KUKA KRL program: EPS_2_251729_MH3A_A_20251114081656.src

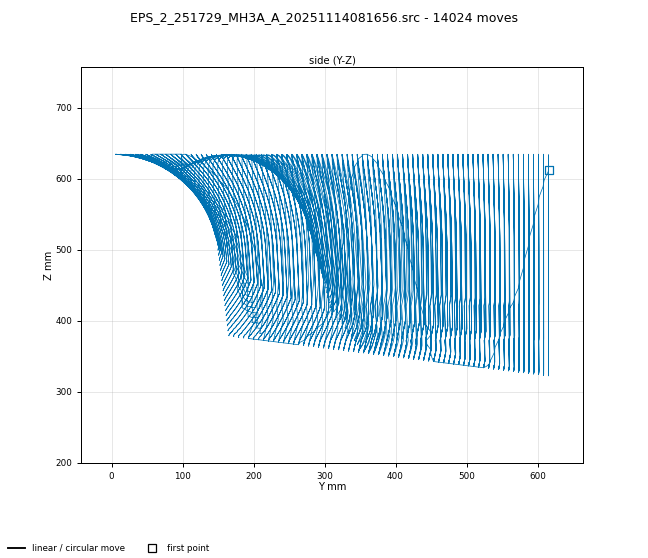
[picture p0: tool path of EPS_2_251729_MH3A_A_20251114081656.src, 14024 of 14026 moves have a stored position in this frame; points joined in program order, loops and branches not executed]
&ACCESS RVP
&REL 4
&COMMENT QRS 19112012
&PARAM EDITMASK = *
DEF PART()
EXT BAS (BAS_COMMAND :IN,REAL :IN )
INT I
BAS (#INITMOV,0 )

;KUKA QRS Post kuka4.cps  Date:22-06-2017 !

File_ID=2916

QRS_PRE_INIT()

;Init var - Until changes are made in qrs_pre_init
Outlet_Square_prg=0
Inlet_1_Square_prg=0
Inlet_2_Square_prg=0
Inlet_3_Square_prg=0
Inlet_4_Square_prg=0
Inlet_5_Square_prg=0

Outlet_1={X 0.000, Y 527.380, Z 509.000, B 0.000, E1 0.000 }
Inlet_1={X 0.000, Y 530.110, Z 534.000, B 0.000, E1 90.000 }
Inlet_2={X 0.000, Y 527.380, Z 509.000, B 0.000, E1 180.000 }
Outlet_1_type=251
Inlet_1_type=201
Inlet_2_type=251
;QRS#1=Sidecore dimensions
;QRS#2=250-10" PVC SDR 35
;QRS#3=200-8" PVC SDR 35
;QRS#4=250-10" PVC SDR 35
;QRS#5=
;QRS#6=
;QRS#7=
;QRS#8=
;QRS#9=14M PSX
;QRS#10=12-08 PSX
;QRS#11=14M PSX
;QRS#12=
;QRS#13=
;QRS#14=
;QRS#15=
;QRS#16=1220x127x914 3'
;QRS#17=EPS Height
;QRS#18=634,5
;QRS#19=*
;QRS#20= UPDATED VERSION 22-06-2017
;QRS#21=*
Outlet_Square=0100
Inlet_1_Square=0100
Inlet_2_Square=0100
Inlet_3_Square=0
Inlet_4_Square=0
Inlet_5_Square=0
Mill_Square=1
Outlet_Square_Prg=205
Inlet_1_Square_prg=204
Inlet_2_Square_prg=205

QRS_INIT()

$ADVANCE=5

; T1
PTP {E1 173.417,E2 173.417}
PTP {X 0,Y 615.497,A -85,B 0,C 180,E1 173.417,E2 173.417,E3 0,E4 0,E5 0,E6 0}
QRS_SPEED_INIT()
LIN {X 0,Y 615.497,Z 612.701,A -85,B 0,C 180,E1 173.417,E2 173.417,E3 0,E4 0,E5 0,E6 0} C_VEL
LIN {X 0,Y 615.497,Z 605.036,A -85,B 0,C 180,E1 172.455,E2 172.455} C_VEL
LIN {X 0,Y 615.498,Z 595.258,A -85,B 0,C 180,E1 171.463,E2 171.463} C_VEL
LIN {X 0,Y 615.497,Z 584.992,A -85,B 0,C 180,E1 170.636,E2 170.636} C_VEL
LIN {X 0,Y 615.479,Z 573.43,A -85,B 0,C 180,E1 169.888,E2 169.888} C_VEL
LIN {X 0,Y 615.499,Z 561.522,A -85,B 0,C 180,E1 169.291,E2 169.291} C_VEL
LIN {X 0,Y 615.498,Z 548.655,A -85,B 0,C 180,E1 168.807,E2 168.807} C_VEL
LIN {X 0,Y 615.493,Z 536.054,A -85,B 0,C 180,E1 168.473,E2 168.473} C_VEL
LIN {X 0,Y 615.488,Z 522.928,A -85,B 0,C 180,E1 168.264,E2 168.264} C_VEL
LIN {X 0,Y 615.497,Z 421.645,A -85,B 0,C 180,E1 167.072,E2 167.072} C_VEL
LIN {X 0,Y 615.491,Z 420.224,A -85,B 0,C 180,E1 166.967,E2 166.967} C_VEL
LIN {X 0,Y 615.492,Z 395.066,A -85,B 0,C 180,E1 164.095,E2 164.095} C_VEL
LIN {X 0,Y 615.492,Z 371.363,A -85,B 0,C 180,E1 161.354,E2 161.354} C_VEL
LIN {X 0,Y 615.498,Z 347.631,A -85,B 0,C 180,E1 158.568,E2 158.568} C_VEL
LIN {X 0,Y 615.497,Z 323.889,A -85,B 0,C 180,E1 155.728,E2 155.728} C_VEL
LIN {X 0,Y 615.495,Z 322.471,A -85,B 0,C 180,E1 155.504,E2 155.504} C_VEL
LIN {X 0,Y 615.484,Z 322.311,A -85,B 0,C 180,E1 152.823,E2 152.823} C_VEL
LIN {X 0,Y 615.477,Z 322.312,A -85,B 0,C 180,E1 150.208,E2 150.208} C_VEL
LIN {X 0,Y 615.495,Z 322.325,A -85,B 0,C 180,E1 147.543,E2 147.543} C_VEL
LIN {X 0,Y 615.481,Z 322.316,A -85,B 0,C 180,E1 145.184,E2 145.184} C_VEL
LIN {X 0,Y 615.489,Z 322.307,A -85,B 0,C 180,E1 142.758,E2 142.758} C_VEL
LIN {X 0,Y 615.485,Z 322.321,A -85,B 0,C 180,E1 139.912,E2 139.912} C_VEL
LIN {X 0,Y 615.491,Z 322.323,A -85,B 0,C 180,E1 137.647,E2 137.647} C_VEL
LIN {X 0,Y 615.48,Z 322.31,A -85,B 0,C 180,E1 134.931,E2 134.931} C_VEL
LIN {X 0,Y 615.485,Z 322.32,A -85,B 0,C 180,E1 132.08,E2 132.08} C_VEL
LIN {X 0,Y 615.494,Z 322.321,A -85,B 0,C 180,E1 129.75,E2 129.75} C_VEL
LIN {X 0,Y 615.483,Z 322.309,A -85,B 0,C 180,E1 126.936,E2 126.936} C_VEL
LIN {X 0,Y 615.494,Z 322.326,A -85,B 0,C 180,E1 124.022,E2 124.022} C_VEL
LIN {X 0,Y 615.488,Z 322.316,A -85,B 0,C 180,E1 121.686,E2 121.686} C_VEL
LIN {X 0,Y 615.477,Z 322.312,A -85,B 0,C 180,E1 119.407,E2 119.407} C_VEL
LIN {X 0,Y 615.486,Z 322.308,A -85,B 0,C 180,E1 117.044,E2 117.044} C_VEL
LIN {X 0,Y 615.491,Z 322.324,A -85,B 0,C 180,E1 114.273,E2 114.273} C_VEL
LIN {X 0,Y 615.495,Z 322.53,A -85,B 0,C 180,E1 112.137,E2 112.137} C_VEL
LIN {X 0,Y 615.495,Z 339.273,A -85,B 0,C 180,E1 109.859,E2 109.859} C_VEL
LIN {X 0,Y 615.493,Z 361.461,A -85,B 0,C 180,E1 106.929,E2 106.929} C_VEL
LIN {X 0,Y 615.479,Z 372.134,A -85,B 0,C 180,E1 105.566,E2 105.566} C_VEL
LIN {X 0,Y 615.477,Z 377.127,A -85,B 0,C 180,E1 105.481,E2 105.481} C_VEL
LIN {X 0,Y 615.498,Z 509.136,A -85,B 0,C 180,E1 103.905,E2 103.905} C_VEL
LIN {X 0,Y 615.497,Z 522.72,A -85,B 0,C 180,E1 103.622,E2 103.622} C_VEL
LIN {X 0,Y 615.497,Z 536.468,A -85,B 0,C 180,E1 103.202,E2 103.202} C_VEL
LIN {X 0,Y 615.493,Z 548.884,A -85,B 0,C 180,E1 102.698,E2 102.698} C_VEL
LIN {X 0,Y 615.496,Z 561.829,A -85,B 0,C 180,E1 102.029,E2 102.029} C_VEL
LIN {X 0,Y 615.499,Z 573.548,A -85,B 0,C 180,E1 101.277,E2 101.277} C_VEL
LIN {X 0,Y 615.498,Z 585.217,A -85,B 0,C 180,E1 100.361,E2 100.361} C_VEL
LIN {X 0,Y 615.497,Z 595.643,A -85,B 0,C 180,E1 99.365,E2 99.365} C_VEL
LIN {X 0,Y 615.496,Z 604.233,A -85,B 0,C 180,E1 98.372,E2 98.372} C_VEL
LIN {X 0,Y 615.495,Z 612.448,A -85,B 0,C 180,E1 97.216,E2 97.216} C_VEL
LIN {X 0,Y 615.496,Z 618.179,A -85,B 0,C 180,E1 96.228,E2 96.228} C_VEL
LIN {X 0,Y 615.491,Z 622.885,A -85,B 0,C 180,E1 95.242,E2 95.242} C_VEL
LIN {X 0,Y 615.496,Z 627.754,A -85,B 0,C 180,E1 93.929,E2 93.929} C_VEL
LIN {X 0,Y 615.496,Z 631.152,A -85,B 0,C 180,E1 92.619,E2 92.619} C_VEL
LIN {X 0,Y 615.493,Z 633.173,A -85,B 0,C 180,E1 91.309,E2 91.309} C_VEL
LIN {X 0,Y 615.494,Z 633.884,A -85,B 0,C 180,E1 90.001,E2 90.001} C_VEL
LIN {X 0,Y 615.49,Z 633.281,A -85,B 0,C 180,E1 88.692,E2 88.692} C_VEL
LIN {X 0,Y 615.493,Z 631.352,A -85,B 0,C 180,E1 87.383,E2 87.383} C_VEL
LIN {X 0,Y 615.496,Z 628.048,A -85,B 0,C 180,E1 86.072,E2 86.072} C_VEL
LIN {X 0,Y 615.496,Z 623.277,A -85,B 0,C 180,E1 84.76,E2 84.76} C_VEL
LIN {X 0,Y 615.494,Z 616.879,A -85,B 0,C 180,E1 83.444,E2 83.444} C_VEL
LIN {X 0,Y 615.496,Z 609.75,A -85,B 0,C 180,E1 82.29,E2 82.29} C_VEL
LIN {X 0,Y 615.497,Z 602.278,A -85,B 0,C 180,E1 81.299,E2 81.299} C_VEL
LIN {X 0,Y 615.495,Z 593.3,A -85,B 0,C 180,E1 80.305,E2 80.305} C_VEL
LIN {X 0,Y 615.499,Z 582.211,A -85,B 0,C 180,E1 79.291,E2 79.291} C_VEL
LIN {X 0,Y 615.498,Z 571.294,A -85,B 0,C 180,E1 78.474,E2 78.474} C_VEL
LIN {X 0,Y 615.489,Z 559,A -85,B 0,C 180,E1 77.722,E2 77.722} C_VEL
LIN {X 0,Y 615.498,Z 547.167,A -85,B 0,C 180,E1 77.136,E2 77.136} C_VEL
LIN {X 0,Y 615.493,Z 534.248,A -85,B 0,C 180,E1 76.632,E2 76.632} C_VEL
LIN {X 0,Y 615.498,Z 521.28,A -85,B 0,C 180,E1 76.253,E2 76.253} C_VEL
LIN {X 0,Y 615.497,Z 507.999,A -85,B 0,C 180,E1 75.988,E2 75.988} C_VEL
LIN {X 0,Y 615.481,Z 372.767,A -85,B 0,C 180,E1 74.372,E2 74.372} C_VEL
LIN {X 0,Y 615.486,Z 371.322,A -85,B 0,C 180,E1 74.266,E2 74.266} C_VEL
LIN {X 0,Y 615.477,Z 350.657,A -85,B 0,C 180,E1 71.559,E2 71.559} C_VEL
LIN {X 0,Y 615.493,Z 329.507,A -85,B 0,C 180,E1 68.745,E2 68.745} C_VEL
LIN {X 0,Y 615.494,Z 322.495,A -85,B 0,C 180,E1 67.759,E2 67.759} C_VEL
LIN {X 0,Y 615.488,Z 322.309,A -85,B 0,C 180,E1 65.009,E2 65.009} C_VEL
LIN {X 0,Y 615.48,Z 322.309,A -85,B 0,C 180,E1 62.824,E2 62.824} C_VEL
LIN {X 0,Y 615.497,Z 322.313,A -85,B 0,C 180,E1 60.204,E2 60.204} C_VEL
LIN {X 0,Y 615.489,Z 322.316,A -85,B 0,C 180,E1 57.544,E2 57.544} C_VEL
LIN {X 0,Y 615.499,Z 322.306,A -85,B 0,C 180,E1 55.187,E2 55.187} C_VEL
LIN {X 0,Y 615.477,Z 322.311,A -85,B 0,C 180,E1 52.759,E2 52.759} C_VEL
LIN {X 0,Y 615.493,Z 322.322,A -85,B 0,C 180,E1 49.911,E2 49.911} C_VEL
LIN {X 0,Y 615.481,Z 322.309,A -85,B 0,C 180,E1 46.953,E2 46.953} C_VEL
LIN {X 0,Y 615.486,Z 322.323,A -85,B 0,C 180,E1 43.999,E2 43.999} C_VEL
LIN {X 0,Y 615.487,Z 322.309,A -85,B 0,C 180,E1 41.474,E2 41.474} C_VEL
LIN {X 0,Y 615.478,Z 322.312,A -85,B 0,C 180,E1 38.905,E2 38.905} C_VEL
LIN {X 0,Y 615.489,Z 322.322,A -85,B 0,C 180,E1 36.425,E2 36.425} C_VEL
LIN {X 0,Y 615.484,Z 322.309,A -85,B 0,C 180,E1 33.536,E2 33.536} C_VEL
LIN {X 0,Y 615.48,Z 322.314,A -85,B 0,C 180,E1 30.92,E2 30.92} C_VEL
LIN {X 0,Y 615.498,Z 322.325,A -85,B 0,C 180,E1 28.455,E2 28.455} C_VEL
LIN {X 0,Y 615.484,Z 322.308,A -85,B 0,C 180,E1 25.571,E2 25.571} C_VEL
LIN {X 0,Y 615.484,Z 322.318,A -85,B 0,C 180,E1 22.845,E2 22.845} C_VEL
LIN {X 0,Y 615.479,Z 322.313,A -85,B 0,C 180,E1 20.033,E2 20.033} C_VEL
LIN {X 0,Y 615.493,Z 322.309,A -85,B 0,C 180,E1 17.27,E2 17.27} C_VEL
LIN {X 0,Y 615.496,Z 322.32,A -85,B 0,C 180,E1 14.549,E2 14.549} C_VEL
LIN {X 0,Y 615.476,Z 322.311,A -85,B 0,C 180,E1 11.861,E2 11.861} C_VEL
LIN {X 0,Y 615.487,Z 322.315,A -85,B 0,C 180,E1 9.199,E2 9.199} C_VEL
LIN {X 0,Y 615.498,Z 322.315,A -85,B 0,C 180,E1 6.557,E2 6.557} C_VEL
LIN {X 0,Y 615.476,Z 322.31,A -85,B 0,C 180,E1 3.929,E2 3.929} C_VEL
LIN {X 0,Y 615.494,Z 322.315,A -85,B 0,C 180,E1 1.309,E2 1.309} C_VEL
LIN {X 0,Y 615.495,Z 322.316,A -85,B 0,C 180,E1 -1.309,E2 -1.309} C_VEL
LIN {X 0,Y 615.476,Z 322.31,A -85,B 0,C 180,E1 -3.929,E2 -3.929} C_VEL
LIN {X 0,Y 615.496,Z 322.316,A -85,B 0,C 180,E1 -6.597,E2 -6.597} C_VEL
LIN {X 0,Y 615.488,Z 322.316,A -85,B 0,C 180,E1 -9.199,E2 -9.199} C_VEL
LIN {X 0,Y 615.478,Z 322.31,A -85,B 0,C 180,E1 -11.861,E2 -11.861} C_VEL
LIN {X 0,Y 615.497,Z 322.319,A -85,B 0,C 180,E1 -14.549,E2 -14.549} C_VEL
LIN {X 0,Y 615.493,Z 322.31,A -85,B 0,C 180,E1 -17.27,E2 -17.27} C_VEL
LIN {X 0,Y 615.479,Z 322.313,A -85,B 0,C 180,E1 -20.033,E2 -20.033} C_VEL
LIN {X 0,Y 615.487,Z 322.319,A -85,B 0,C 180,E1 -22.845,E2 -22.845} C_VEL
LIN {X 0,Y 615.484,Z 322.308,A -85,B 0,C 180,E1 -25.571,E2 -25.571} C_VEL
LIN {X 0,Y 615.497,Z 322.325,A -85,B 0,C 180,E1 -28.455,E2 -28.455} C_VEL
LIN {X 0,Y 615.486,Z 322.31,A -85,B 0,C 180,E1 -31.088,E2 -31.088} C_VEL
LIN {X 0,Y 615.484,Z 322.309,A -85,B 0,C 180,E1 -33.536,E2 -33.536} C_VEL
LIN {X 0,Y 615.488,Z 322.324,A -85,B 0,C 180,E1 -36.425,E2 -36.425} C_VEL
LIN {X 0,Y 615.481,Z 322.31,A -85,B 0,C 180,E1 -39.063,E2 -39.063} C_VEL
LIN {X 0,Y 615.486,Z 322.309,A -85,B 0,C 180,E1 -41.474,E2 -41.474} C_VEL
LIN {X 0,Y 615.497,Z 322.325,A -85,B 0,C 180,E1 -44.149,E2 -44.149} C_VEL
LIN {X 0,Y 615.481,Z 322.31,A -85,B 0,C 180,E1 -46.953,E2 -46.953} C_VEL
LIN {X 0,Y 615.485,Z 322.31,A -85,B 0,C 180,E1 -49.395,E2 -49.395} C_VEL
LIN {X 0,Y 615.49,Z 322.326,A -85,B 0,C 180,E1 -51.988,E2 -51.988} C_VEL
LIN {X 0,Y 615.486,Z 322.315,A -85,B 0,C 180,E1 -54.385,E2 -54.385} C_VEL
LIN {X 0,Y 615.478,Z 322.31,A -85,B 0,C 180,E1 -56.765,E2 -56.765} C_VEL
LIN {X 0,Y 615.492,Z 322.307,A -85,B 0,C 180,E1 -59.082,E2 -59.082} C_VEL
LIN {X 0,Y 615.489,Z 322.317,A -85,B 0,C 180,E1 -61.55,E2 -61.55} C_VEL
LIN {X 0,Y 615.481,Z 322.312,A -85,B 0,C 180,E1 -64.433,E2 -64.433} C_VEL
LIN {X 0,Y 615.49,Z 322.311,A -85,B 0,C 180,E1 -67.157,E2 -67.157} C_VEL
LIN {X 0,Y 615.494,Z 322.613,A -85,B 0,C 180,E1 -67.838,E2 -67.838} C_VEL
LIN {X 0,Y 615.491,Z 340.931,A -85,B 0,C 180,E1 -70.316,E2 -70.316} C_VEL
LIN {X 0,Y 615.493,Z 361.818,A -85,B 0,C 180,E1 -73.073,E2 -73.073} C_VEL
LIN {X 0,Y 615.481,Z 371.9,A -85,B 0,C 180,E1 -74.372,E2 -74.372} C_VEL
LIN {X 0,Y 615.479,Z 373.911,A -85,B 0,C 180,E1 -74.435,E2 -74.435} C_VEL
LIN {X 0,Y 615.5,Z 509.9,A -85,B 0,C 180,E1 -76.063,E2 -76.063} C_VEL
LIN {X 0,Y 615.497,Z 524.411,A -85,B 0,C 180,E1 -76.38,E2 -76.38} C_VEL
LIN {X 0,Y 615.497,Z 537.713,A -85,B 0,C 180,E1 -76.8,E2 -76.8} C_VEL
LIN {X 0,Y 615.497,Z 549.856,A -85,B 0,C 180,E1 -77.303,E2 -77.303} C_VEL
LIN {X 0,Y 615.493,Z 562.615,A -85,B 0,C 180,E1 -77.973,E2 -77.973} C_VEL
LIN {X 0,Y 615.499,Z 575.353,A -85,B 0,C 180,E1 -78.808,E2 -78.808} C_VEL
LIN {X 0,Y 615.498,Z 585.759,A -85,B 0,C 180,E1 -79.641,E2 -79.641} C_VEL
LIN {X 0,Y 615.496,Z 596.097,A -85,B 0,C 180,E1 -80.637,E2 -80.637} C_VEL
LIN {X 0,Y 615.497,Z 604.61,A -85,B 0,C 180,E1 -81.63,E2 -81.63} C_VEL
LIN {X 0,Y 615.496,Z 612.732,A -85,B 0,C 180,E1 -82.785,E2 -82.785} C_VEL
LIN {X 0,Y 615.496,Z 618.435,A -85,B 0,C 180,E1 -83.773,E2 -83.773} C_VEL
LIN {X 0,Y 615.495,Z 623.084,A -85,B 0,C 180,E1 -84.76,E2 -84.76} C_VEL
LIN {X 0,Y 615.494,Z 627.904,A -85,B 0,C 180,E1 -86.072,E2 -86.072} C_VEL
LIN {X 0,Y 615.496,Z 631.254,A -85,B 0,C 180,E1 -87.383,E2 -87.383} C_VEL
LIN {X 0,Y 615.489,Z 633.23,A -85,B 0,C 180,E1 -88.692,E2 -88.692} C_VEL
LIN {X 0,Y 615.493,Z 633.889,A -85,B 0,C 180,E1 -90.001,E2 -90.001} C_VEL
LIN {X 0,Y 615.489,Z 633.228,A -85,B 0,C 180,E1 -91.309,E2 -91.309} C_VEL
LIN {X 0,Y 615.496,Z 631.25,A -85,B 0,C 180,E1 -92.619,E2 -92.619} C_VEL
LIN {X 0,Y 615.494,Z 627.899,A -85,B 0,C 180,E1 -93.929,E2 -93.929} C_VEL
LIN {X 0,Y 615.495,Z 623.077,A -85,B 0,C 180,E1 -95.242,E2 -95.242} C_VEL
LIN {X 0,Y 615.496,Z 616.624,A -85,B 0,C 180,E1 -96.557,E2 -96.557} C_VEL
LIN {X 0,Y 615.497,Z 609.435,A -85,B 0,C 180,E1 -97.711,E2 -97.711} C_VEL
LIN {X 0,Y 615.497,Z 601.897,A -85,B 0,C 180,E1 -98.703,E2 -98.703} C_VEL
LIN {X 0,Y 615.495,Z 592.845,A -85,B 0,C 180,E1 -99.697,E2 -99.697} C_VEL
LIN {X 0,Y 615.497,Z 582.751,A -85,B 0,C 180,E1 -100.619,E2 -100.619} C_VEL
LIN {X 0,Y 615.498,Z 571.846,A -85,B 0,C 180,E1 -101.444,E2 -101.444} C_VEL
LIN {X 0,Y 615.488,Z 559.691,A -85,B 0,C 180,E1 -102.196,E2 -102.196} C_VEL
LIN {X 0,Y 615.498,Z 546.072,A -85,B 0,C 180,E1 -102.866,E2 -102.866} C_VEL
LIN {X 0,Y 615.497,Z 532.811,A -85,B 0,C 180,E1 -103.37,E2 -103.37} C_VEL
LIN {X 0,Y 615.498,Z 519.253,A -85,B 0,C 180,E1 -103.748,E2 -103.748} C_VEL
LIN {X 0,Y 615.497,Z 504.746,A -85,B 0,C 180,E1 -104.013,E2 -104.013} C_VEL
LIN {X 0,Y 615.48,Z 372.617,A -85,B 0,C 180,E1 -105.587,E2 -105.587} C_VEL
LIN {X 0,Y 615.486,Z 370.938,A -85,B 0,C 180,E1 -105.736,E2 -105.736} C_VEL
LIN {X 0,Y 615.477,Z 350.311,A -85,B 0,C 180,E1 -108.441,E2 -108.441} C_VEL
LIN {X 0,Y 615.496,Z 329.159,A -85,B 0,C 180,E1 -111.257,E2 -111.257} C_VEL
LIN {X 0,Y 615.494,Z 322.512,A -85,B 0,C 180,E1 -112.189,E2 -112.189} C_VEL
LIN {X 0,Y 615.492,Z 322.325,A -85,B 0,C 180,E1 -114.272,E2 -114.272} C_VEL
LIN {X 0,Y 615.486,Z 322.308,A -85,B 0,C 180,E1 -117.045,E2 -117.045} C_VEL
LIN {X 0,Y 615.497,Z 322.314,A -85,B 0,C 180,E1 -119.796,E2 -119.796} C_VEL
LIN {X 0,Y 615.488,Z 322.316,A -85,B 0,C 180,E1 -122.458,E2 -122.458} C_VEL
LIN {X 0,Y 615.499,Z 322.306,A -85,B 0,C 180,E1 -124.815,E2 -124.815} C_VEL
LIN {X 0,Y 615.477,Z 322.311,A -85,B 0,C 180,E1 -127.244,E2 -127.244} C_VEL
LIN {X 0,Y 615.492,Z 322.322,A -85,B 0,C 180,E1 -130.089,E2 -130.089} C_VEL
LIN {X 0,Y 615.481,Z 322.309,A -85,B 0,C 180,E1 -133.047,E2 -133.047} C_VEL
LIN {X 0,Y 615.486,Z 322.323,A -85,B 0,C 180,E1 -136.003,E2 -136.003} C_VEL
LIN {X 0,Y 615.487,Z 322.309,A -85,B 0,C 180,E1 -138.526,E2 -138.526} C_VEL
LIN {X 0,Y 615.478,Z 322.312,A -85,B 0,C 180,E1 -141.095,E2 -141.095} C_VEL
LIN {X 0,Y 615.489,Z 322.322,A -85,B 0,C 180,E1 -143.575,E2 -143.575} C_VEL
LIN {X 0,Y 615.484,Z 322.309,A -85,B 0,C 180,E1 -146.467,E2 -146.467} C_VEL
LIN {X 0,Y 615.48,Z 322.313,A -85,B 0,C 180,E1 -149.08,E2 -149.08} C_VEL
LIN {X 0,Y 615.497,Z 322.324,A -85,B 0,C 180,E1 -151.549,E2 -151.549} C_VEL
LIN {X 0,Y 615.484,Z 322.308,A -85,B 0,C 180,E1 -154.433,E2 -154.433} C_VEL
LIN {X 0,Y 615.499,Z 322.572,A -85,B 0,C 180,E1 -155.639,E2 -155.639} C_VEL
LIN {X 0,Y 615.479,Z 343.906,A -85,B 0,C 180,E1 -158.216,E2 -158.216} C_VEL
LIN {X 0,Y 615.484,Z 367.627,A -85,B 0,C 180,E1 -161.008,E2 -161.008} C_VEL
LIN {X 0,Y 615.483,Z 391.999,A -85,B 0,C 180,E1 -163.832,E2 -163.832} C_VEL
LIN {X 0,Y 615.491,Z 416.465,A -85,B 0,C 180,E1 -166.631,E2 -166.631} C_VEL
LIN {X 0,Y 615.495,Z 421.071,A -85,B 0,C 180,E1 -167.135,E2 -167.135} C_VEL
LIN {X 0,Y 615.491,Z 425.922,A -85,B 0,C 180,E1 -167.219,E2 -167.219} C_VEL
LIN {X 0,Y 615.486,Z 530.146,A -85,B 0,C 180,E1 -168.452,E2 -168.452} C_VEL
LIN {X 0,Y 615.499,Z 542.722,A -85,B 0,C 180,E1 -168.724,E2 -168.724} C_VEL
LIN {X 0,Y 615.497,Z 556.026,A -85,B 0,C 180,E1 -169.155,E2 -169.155} C_VEL
LIN {X 0,Y 615.491,Z 567.066,A -85,B 0,C 180,E1 -169.639,E2 -169.639} C_VEL
LIN {X 0,Y 615.482,Z 578.806,A -85,B 0,C 180,E1 -170.304,E2 -170.304} C_VEL
LIN {X 0,Y 615.499,Z 589.268,A -85,B 0,C 180,E1 -171.05,E2 -171.05} C_VEL
LIN {X 0,Y 615.498,Z 597.831,A -85,B 0,C 180,E1 -171.794,E2 -171.794} C_VEL
LIN {X 0,Y 615.498,Z 605.709,A -85,B 0,C 180,E1 -172.62,E2 -172.62} C_VEL
LIN {X 0,Y 615.497,Z 613.399,A -85,B 0,C 180,E1 -173.608,E2 -173.608} C_VEL
LIN {X 0,Y 615.498,Z 620.458,A -85,B 0,C 180,E1 -174.759,E2 -174.759} C_VEL
LIN {X 0,Y 615.493,Z 625.158,A -85,B 0,C 180,E1 -175.744,E2 -175.744} C_VEL
LIN {X 0,Y 615.496,Z 628.754,A -85,B 0,C 180,E1 -176.727,E2 -176.727} C_VEL
LIN {X 0,Y 615.496,Z 630.615,A -85,B 0,C 180,E1 -177.382,E2 -177.382} C_VEL
LIN {X 0,Y 615.497,Z 632.034,A -85,B 0,C 180,E1 -178.037,E2 -178.037} C_VEL
LIN {X 0,Y 615.496,Z 633.642,A -85,B 0,C 180,E1 -179.346,E2 -179.346} C_VEL
LIN {X 0,Y 615.494,Z 633.884,A -85,B 0,C 180,E1 -180,E2 -180} C_VEL
LIN {X 0,Y 615.496,Z 633.705,A -85,B 0,C 180,E1 -180.654,E2 -180.654} C_VEL
LIN {X 0,Y 615.496,Z 632.183,A -85,B 0,C 180,E1 -181.963,E2 -181.963} C_VEL
LIN {X 0,Y 615.498,Z 630.841,A -85,B 0,C 180,E1 -182.618,E2 -182.618} C_VEL
LIN {X 0,Y 615.497,Z 627.994,A -85,B 0,C 180,E1 -183.601,E2 -183.601} C_VEL
LIN {X 0,Y 615.499,Z 624.134,A -85,B 0,C 180,E1 -184.585,E2 -184.585} C_VEL
LIN {X 0,Y 615.498,Z 619.151,A -85,B 0,C 180,E1 -185.57,E2 -185.57} C_VEL
LIN {X 0,Y 615.497,Z 612.701,A -85,B 0,C 180,E1 -186.583,E2 -186.583} C_VEL
LIN {X 0,Y 614.829,Z 609.519,A -85,B 0,C 180,E1 -187.032,E2 -187.032} C_VEL
LIN {X 0,Y 611.988,Z 603.946,A -85,B 0,C 180,E1 -187.749,E2 -187.749} C_VEL
LIN {X 0,Y 609.138,Z 597.67,A -85,B 0,C 180,E1 -188.43,E2 -188.43} C_VEL
LIN {X 0,Y 608.477,Z 593.429,A -85,B 0,C 180,E1 -188.82,E2 -188.82} C_VEL
LIN {X 0,Y 608.489,Z 582.891,A -85,B 0,C 180,E1 -189.641,E2 -189.641} C_VEL
LIN {X 0,Y 608.49,Z 572.112,A -85,B 0,C 180,E1 -190.313,E2 -190.313} C_VEL
LIN {X 0,Y 608.515,Z 560.848,A -85,B 0,C 180,E1 -190.868,E2 -190.868} C_VEL
LIN {X 0,Y 608.534,Z 548.763,A -85,B 0,C 180,E1 -191.323,E2 -191.323} C_VEL
LIN {X 0,Y 608.542,Z 536.148,A -85,B 0,C 180,E1 -191.66,E2 -191.66} C_VEL
LIN {X 0,Y 608.539,Z 523.034,A -85,B 0,C 180,E1 -191.871,E2 -191.871} C_VEL
LIN {X 0,Y 608.556,Z 421.658,A -85,B 0,C 180,E1 -193.078,E2 -193.078} C_VEL
LIN {X 0,Y 608.48,Z 420.328,A -85,B 0,C 180,E1 -193.186,E2 -193.186} C_VEL
LIN {X 0,Y 608.533,Z 396.59,A -85,B 0,C 180,E1 -195.92,E2 -195.92} C_VEL
LIN {X 0,Y 608.546,Z 372.479,A -85,B 0,C 180,E1 -198.736,E2 -198.736} C_VEL
LIN {X 0,Y 608.623,Z 349.11,A -85,B 0,C 180,E1 -201.508,E2 -201.508} C_VEL
LIN {X 0,Y 608.674,Z 324.899,A -85,B 0,C 180,E1 -204.437,E2 -204.437} C_VEL
LIN {X 0,Y 608.49,Z 323.441,A -85,B 0,C 180,E1 -204.661,E2 -204.661} C_VEL
LIN {X 0,Y 608.447,Z 323.313,A -85,B 0,C 180,E1 -207.518,E2 -207.518} C_VEL
LIN {X 0,Y 608.462,Z 323.314,A -85,B 0,C 180,E1 -209.97,E2 -209.97} C_VEL
LIN {X 0,Y 608.463,Z 323.314,A -85,B 0,C 180,E1 -212.879,E2 -212.879} C_VEL
LIN {X 0,Y 608.439,Z 323.314,A -85,B 0,C 180,E1 -215.278,E2 -215.278} C_VEL
LIN {X 0,Y 608.468,Z 323.312,A -85,B 0,C 180,E1 -217.746,E2 -217.746} C_VEL
LIN {X 0,Y 608.448,Z 323.323,A -85,B 0,C 180,E1 -220.328,E2 -220.328} C_VEL
LIN {X 0,Y 608.484,Z 323.308,A -85,B 0,C 180,E1 -223.31,E2 -223.31} C_VEL
LIN {X 0,Y 608.469,Z 323.32,A -85,B 0,C 180,E1 -226.13,E2 -226.13} C_VEL
LIN {X 0,Y 608.45,Z 323.314,A -85,B 0,C 180,E1 -228.822,E2 -228.822} C_VEL
LIN {X 0,Y 608.469,Z 323.315,A -85,B 0,C 180,E1 -231.76,E2 -231.76} C_VEL
LIN {X 0,Y 608.449,Z 323.314,A -85,B 0,C 180,E1 -234.722,E2 -234.722} C_VEL
LIN {X 0,Y 608.462,Z 323.314,A -85,B 0,C 180,E1 -237.478,E2 -237.478} C_VEL
LIN {X 0,Y 608.481,Z 323.314,A -85,B 0,C 180,E1 -240.221,E2 -240.221} C_VEL
LIN {X 0,Y 608.477,Z 323.31,A -85,B 0,C 180,E1 -242.794,E2 -242.794} C_VEL
LIN {X 0,Y 608.457,Z 323.316,A -85,B 0,C 180,E1 -245.428,E2 -245.428} C_VEL
LIN {X 0,Y 608.493,Z 323.473,A -85,B 0,C 180,E1 -247.729,E2 -247.729} C_VEL
LIN {X 0,Y 608.574,Z 331.445,A -85,B 0,C 180,E1 -248.845,E2 -248.845} C_VEL
LIN {X 0,Y 608.511,Z 352.446,A -85,B 0,C 180,E1 -251.666,E2 -251.666} C_VEL
LIN {X 0,Y 608.531,Z 372.139,A -85,B 0,C 180,E1 -254.251,E2 -254.251} C_VEL
LIN {X 0,Y 608.647,Z 375.384,A -85,B 0,C 180,E1 -254.319,E2 -254.319} C_VEL
LIN {X 0,Y 608.61,Z 509.953,A -85,B 0,C 180,E1 -255.948,E2 -255.948} C_VEL
LIN {X 0,Y 608.613,Z 524.281,A -85,B 0,C 180,E1 -256.263,E2 -256.263} C_VEL
LIN {X 0,Y 608.586,Z 537.623,A -85,B 0,C 180,E1 -256.688,E2 -256.688} C_VEL
LIN {X 0,Y 608.544,Z 550.675,A -85,B 0,C 180,E1 -257.239,E2 -257.239} C_VEL
LIN {X 0,Y 608.536,Z 563.327,A -85,B 0,C 180,E1 -257.916,E2 -257.916} C_VEL
LIN {X 0,Y 608.5,Z 574.843,A -85,B 0,C 180,E1 -258.676,E2 -258.676} C_VEL
LIN {X 0,Y 608.495,Z 585.406,A -85,B 0,C 180,E1 -259.518,E2 -259.518} C_VEL
LIN {X 0,Y 608.48,Z 595.892,A -85,B 0,C 180,E1 -260.526,E2 -260.526} C_VEL
LIN {X 0,Y 608.463,Z 604.543,A -85,B 0,C 180,E1 -261.531,E2 -261.531} C_VEL
LIN {X 0,Y 608.461,Z 612.834,A -85,B 0,C 180,E1 -262.7,E2 -262.7} C_VEL
LIN {X 0,Y 608.443,Z 619.323,A -85,B 0,C 180,E1 -263.831,E2 -263.831} C_VEL
LIN {X 0,Y 608.437,Z 624.784,A -85,B 0,C 180,E1 -265.029,E2 -265.029} C_VEL
LIN {X 0,Y 608.434,Z 628.296,A -85,B 0,C 180,E1 -266.025,E2 -266.025} C_VEL
LIN {X 0,Y 608.424,Z 631.732,A -85,B 0,C 180,E1 -267.351,E2 -267.351} C_VEL
LIN {X 0,Y 608.446,Z 633.776,A -85,B 0,C 180,E1 -268.675,E2 -268.675} C_VEL
LIN {X 0,Y 608.434,Z 634.495,A -85,B 0,C 180,E1 -269.999,E2 -269.999} C_VEL
LIN {X 0,Y 608.443,Z 633.883,A -85,B 0,C 180,E1 -271.323,E2 -271.323} C_VEL
LIN {X 0,Y 608.421,Z 631.93,A -85,B 0,C 180,E1 -272.647,E2 -272.647} C_VEL
LIN {X 0,Y 608.434,Z 628.588,A -85,B 0,C 180,E1 -273.973,E2 -273.973} C_VEL
LIN {X 0,Y 608.44,Z 623.765,A -85,B 0,C 180,E1 -275.301,E2 -275.301} C_VEL
LIN {X 0,Y 608.438,Z 617.301,A -85,B 0,C 180,E1 -276.632,E2 -276.632} C_VEL
LIN {X 0,Y 608.453,Z 610.103,A -85,B 0,C 180,E1 -277.799,E2 -277.799} C_VEL
LIN {X 0,Y 608.476,Z 602.569,A -85,B 0,C 180,E1 -278.802,E2 -278.802} C_VEL
LIN {X 0,Y 608.486,Z 593.528,A -85,B 0,C 180,E1 -279.808,E2 -279.808} C_VEL
LIN {X 0,Y 608.507,Z 582.723,A -85,B 0,C 180,E1 -280.804,E2 -280.804} C_VEL
LIN {X 0,Y 608.523,Z 571.394,A -85,B 0,C 180,E1 -281.66,E2 -281.66} C_VEL
LIN {X 0,Y 608.54,Z 559.061,A -85,B 0,C 180,E1 -282.42,E2 -282.42} C_VEL
LIN {X 0,Y 608.56,Z 547.196,A -85,B 0,C 180,E1 -283.013,E2 -283.013} C_VEL
LIN {X 0,Y 608.581,Z 534.246,A -85,B 0,C 180,E1 -283.523,E2 -283.523} C_VEL
LIN {X 0,Y 608.593,Z 519.989,A -85,B 0,C 180,E1 -283.935,E2 -283.935} C_VEL
LIN {X 0,Y 608.614,Z 506.662,A -85,B 0,C 180,E1 -284.192,E2 -284.192} C_VEL
LIN {X 0,Y 608.587,Z 372.733,A -85,B 0,C 180,E1 -285.81,E2 -285.81} C_VEL
LIN {X 0,Y 608.498,Z 371.369,A -85,B 0,C 180,E1 -285.92,E2 -285.92} C_VEL
LIN {X 0,Y 608.524,Z 351.904,A -85,B 0,C 180,E1 -288.495,E2 -288.495} C_VEL
LIN {X 0,Y 608.571,Z 330.813,A -85,B 0,C 180,E1 -291.331,E2 -291.331} C_VEL
LIN {X 0,Y 608.495,Z 323.483,A -85,B 0,C 180,E1 -292.359,E2 -292.359} C_VEL
LIN {X 0,Y 608.457,Z 323.318,A -85,B 0,C 180,E1 -294.57,E2 -294.57} C_VEL
LIN {X 0,Y 608.475,Z 323.31,A -85,B 0,C 180,E1 -297.206,E2 -297.206} C_VEL
LIN {X 0,Y 608.477,Z 323.316,A -85,B 0,C 180,E1 -299.973,E2 -299.973} C_VEL
LIN {X 0,Y 608.463,Z 323.315,A -85,B 0,C 180,E1 -302.522,E2 -302.522} C_VEL
LIN {X 0,Y 608.447,Z 323.314,A -85,B 0,C 180,E1 -305.276,E2 -305.276} C_VEL
LIN {X 0,Y 608.471,Z 323.317,A -85,B 0,C 180,E1 -308.24,E2 -308.24} C_VEL
LIN {X 0,Y 608.477,Z 323.314,A -85,B 0,C 180,E1 -310.332,E2 -310.332} C_VEL
LIN {X 0,Y 608.465,Z 323.313,A -85,B 0,C 180,E1 -313.308,E2 -313.308} C_VEL
LIN {X 0,Y 608.471,Z 323.316,A -85,B 0,C 180,E1 -316.131,E2 -316.131} C_VEL
LIN {X 0,Y 608.452,Z 323.312,A -85,B 0,C 180,E1 -318.823,E2 -318.823} C_VEL
LIN {X 0,Y 608.464,Z 323.315,A -85,B 0,C 180,E1 -321.411,E2 -321.411} C_VEL
LIN {X 0,Y 608.47,Z 323.317,A -85,B 0,C 180,E1 -323.949,E2 -323.949} C_VEL
LIN {X 0,Y 608.46,Z 323.313,A -85,B 0,C 180,E1 -326.329,E2 -326.329} C_VEL
LIN {X 0,Y 608.471,Z 323.31,A -85,B 0,C 180,E1 -328.726,E2 -328.726} C_VEL
LIN {X 0,Y 608.476,Z 323.316,A -85,B 0,C 180,E1 -331.377,E2 -331.377} C_VEL
LIN {X 0,Y 608.445,Z 323.317,A -85,B 0,C 180,E1 -333.964,E2 -333.964} C_VEL
LIN {X 0,Y 608.461,Z 323.313,A -85,B 0,C 180,E1 -336.155,E2 -336.155} C_VEL
LIN {X 0,Y 608.47,Z 323.31,A -85,B 0,C 180,E1 -338.308,E2 -338.308} C_VEL
LIN {X 0,Y 608.471,Z 323.319,A -85,B 0,C 180,E1 -341.28,E2 -341.28} C_VEL
LIN {X 0,Y 608.457,Z 323.314,A -85,B 0,C 180,E1 -343.906,E2 -343.906} C_VEL
LIN {X 0,Y 608.463,Z 323.312,A -85,B 0,C 180,E1 -346.643,E2 -346.643} C_VEL
LIN {X 0,Y 608.474,Z 323.318,A -85,B 0,C 180,E1 -349.35,E2 -349.35} C_VEL
LIN {X 0,Y 608.471,Z 323.31,A -85,B 0,C 180,E1 -352.033,E2 -352.033} C_VEL
LIN {X 0,Y 608.469,Z 323.314,A -85,B 0,C 180,E1 -354.698,E2 -354.698} C_VEL
LIN {X 0,Y 608.485,Z 323.314,A -85,B 0,C 180,E1 -357.352,E2 -357.352} C_VEL
LIN {X 0,Y 608.468,Z 323.311,A -85,B 0,C 180,E1 -360,E2 -360} C_VEL
LIN {X 0,Y 608.485,Z 323.313,A -85,B 0,C 180,E1 -362.648,E2 -362.648} C_VEL
LIN {X 0,Y 608.47,Z 323.314,A -85,B 0,C 180,E1 -365.302,E2 -365.302} C_VEL
LIN {X 0,Y 608.471,Z 323.31,A -85,B 0,C 180,E1 -367.967,E2 -367.967} C_VEL
LIN {X 0,Y 608.473,Z 323.317,A -85,B 0,C 180,E1 -370.65,E2 -370.65} C_VEL
LIN {X 0,Y 608.464,Z 323.313,A -85,B 0,C 180,E1 -373.356,E2 -373.356} C_VEL
LIN {X 0,Y 608.457,Z 323.313,A -85,B 0,C 180,E1 -376.094,E2 -376.094} C_VEL
LIN {X 0,Y 608.455,Z 323.319,A -85,B 0,C 180,E1 -378.87,E2 -378.87} C_VEL
LIN {X 0,Y 608.47,Z 323.31,A -85,B 0,C 180,E1 -381.691,E2 -381.691} C_VEL
LIN {X 0,Y 608.452,Z 323.323,A -85,B 0,C 180,E1 -384.571,E2 -384.571} C_VEL
LIN {X 0,Y 608.475,Z 323.31,A -85,B 0,C 180,E1 -387.209,E2 -387.209} C_VEL
LIN {X 0,Y 608.46,Z 323.314,A -85,B 0,C 180,E1 -389.973,E2 -389.973} C_VEL
LIN {X 0,Y 608.467,Z 323.319,A -85,B 0,C 180,E1 -392.526,E2 -392.526} C_VEL
LIN {X 0,Y 608.437,Z 323.314,A -85,B 0,C 180,E1 -395.278,E2 -395.278} C_VEL
LIN {X 0,Y 608.467,Z 323.312,A -85,B 0,C 180,E1 -397.746,E2 -397.746} C_VEL
LIN {X 0,Y 608.474,Z 323.319,A -85,B 0,C 180,E1 -400.333,E2 -400.333} C_VEL
LIN {X 0,Y 608.483,Z 323.309,A -85,B 0,C 180,E1 -403.312,E2 -403.312} C_VEL
LIN {X 0,Y 608.467,Z 323.321,A -85,B 0,C 180,E1 -406.132,E2 -406.132} C_VEL
LIN {X 0,Y 608.45,Z 323.313,A -85,B 0,C 180,E1 -408.825,E2 -408.825} C_VEL
LIN {X 0,Y 608.47,Z 323.312,A -85,B 0,C 180,E1 -411.414,E2 -411.414} C_VEL
LIN {X 0,Y 608.476,Z 323.32,A -85,B 0,C 180,E1 -413.951,E2 -413.951} C_VEL
LIN {X 0,Y 608.464,Z 323.315,A -85,B 0,C 180,E1 -416.331,E2 -416.331} C_VEL
LIN {X 0,Y 608.474,Z 323.31,A -85,B 0,C 180,E1 -418.728,E2 -418.728} C_VEL
LIN {X 0,Y 608.476,Z 323.312,A -85,B 0,C 180,E1 -421.38,E2 -421.38} C_VEL
LIN {X 0,Y 608.471,Z 323.313,A -85,B 0,C 180,E1 -424.28,E2 -424.28} C_VEL
LIN {X 0,Y 608.45,Z 323.314,A -85,B 0,C 180,E1 -426.877,E2 -426.877} C_VEL
LIN {X 0,Y 608.505,Z 323.481,A -85,B 0,C 180,E1 -427.686,E2 -427.686} C_VEL
LIN {X 0,Y 608.57,Z 335.111,A -85,B 0,C 180,E1 -429.296,E2 -429.296} C_VEL
LIN {X 0,Y 608.546,Z 356.635,A -85,B 0,C 180,E1 -432.18,E2 -432.18} C_VEL
LIN {X 0,Y 608.541,Z 372.196,A -85,B 0,C 180,E1 -434.21,E2 -434.21} C_VEL
LIN {X 0,Y 608.66,Z 375.699,A -85,B 0,C 180,E1 -434.278,E2 -434.278} C_VEL
LIN {X 0,Y 608.62,Z 508.97,A -85,B 0,C 180,E1 -435.886,E2 -435.886} C_VEL
LIN {X 0,Y 608.595,Z 523.658,A -85,B 0,C 180,E1 -436.201,E2 -436.201} C_VEL
LIN {X 0,Y 608.584,Z 537.735,A -85,B 0,C 180,E1 -436.647,E2 -436.647} C_VEL
LIN {X 0,Y 608.564,Z 549.903,A -85,B 0,C 180,E1 -437.156,E2 -437.156} C_VEL
LIN {X 0,Y 608.516,Z 562.696,A -85,B 0,C 180,E1 -437.833,E2 -437.833} C_VEL
LIN {X 0,Y 608.499,Z 575.483,A -85,B 0,C 180,E1 -438.678,E2 -438.678} C_VEL
LIN {X 0,Y 608.495,Z 585.942,A -85,B 0,C 180,E1 -439.52,E2 -439.52} C_VEL
LIN {X 0,Y 608.479,Z 596.343,A -85,B 0,C 180,E1 -440.528,E2 -440.528} C_VEL
LIN {X 0,Y 608.464,Z 604.921,A -85,B 0,C 180,E1 -441.532,E2 -441.532} C_VEL
LIN {X 0,Y 608.461,Z 613.119,A -85,B 0,C 180,E1 -442.701,E2 -442.701} C_VEL
LIN {X 0,Y 608.443,Z 619.548,A -85,B 0,C 180,E1 -443.831,E2 -443.831} C_VEL
LIN {X 0,Y 608.438,Z 624.965,A -85,B 0,C 180,E1 -445.031,E2 -445.031} C_VEL
LIN {X 0,Y 608.431,Z 628.444,A -85,B 0,C 180,E1 -446.027,E2 -446.027} C_VEL
LIN {X 0,Y 608.424,Z 631.833,A -85,B 0,C 180,E1 -447.353,E2 -447.353} C_VEL
LIN {X 0,Y 608.442,Z 633.831,A -85,B 0,C 180,E1 -448.677,E2 -448.677} C_VEL
LIN {X 0,Y 608.433,Z 634.5,A -85,B 0,C 180,E1 -450.001,E2 -450.001} C_VEL
LIN {X 0,Y 608.442,Z 633.829,A -85,B 0,C 180,E1 -451.325,E2 -451.325} C_VEL
LIN {X 0,Y 608.424,Z 631.829,A -85,B 0,C 180,E1 -452.649,E2 -452.649} C_VEL
LIN {X 0,Y 608.431,Z 628.439,A -85,B 0,C 180,E1 -453.975,E2 -453.975} C_VEL
LIN {X 0,Y 608.44,Z 623.564,A -85,B 0,C 180,E1 -455.303,E2 -455.303} C_VEL
LIN {X 0,Y 608.446,Z 617.207,A -85,B 0,C 180,E1 -456.604,E2 -456.604} C_VEL
LIN {X 0,Y 608.453,Z 609.792,A -85,B 0,C 180,E1 -457.801,E2 -457.801} C_VEL
LIN {X 0,Y 608.473,Z 600.816,A -85,B 0,C 180,E1 -458.971,E2 -458.971} C_VEL
LIN {X 0,Y 608.472,Z 591.382,A -85,B 0,C 180,E1 -459.978,E2 -459.978} C_VEL
LIN {X 0,Y 608.506,Z 580.045,A -85,B 0,C 180,E1 -460.973,E2 -460.973} C_VEL
LIN {X 0,Y 608.533,Z 568.136,A -85,B 0,C 180,E1 -461.83,E2 -461.83} C_VEL
LIN {X 0,Y 608.53,Z 555.057,A -85,B 0,C 180,E1 -462.592,E2 -462.592} C_VEL
LIN {X 0,Y 608.563,Z 542.154,A -85,B 0,C 180,E1 -463.185,E2 -463.185} C_VEL
LIN {X 0,Y 608.597,Z 528.154,A -85,B 0,C 180,E1 -463.673,E2 -463.673} C_VEL
LIN {X 0,Y 608.624,Z 514.411,A -85,B 0,C 180,E1 -464.013,E2 -464.013} C_VEL
LIN {X 0,Y 608.624,Z 500.064,A -85,B 0,C 180,E1 -464.235,E2 -464.235} C_VEL
LIN {X 0,Y 608.558,Z 372.624,A -85,B 0,C 180,E1 -465.769,E2 -465.769} C_VEL
LIN {X 0,Y 608.496,Z 371.005,A -85,B 0,C 180,E1 -465.921,E2 -465.921} C_VEL
LIN {X 0,Y 608.524,Z 351.559,A -85,B 0,C 180,E1 -468.496,E2 -468.496} C_VEL
LIN {X 0,Y 608.574,Z 330.469,A -85,B 0,C 180,E1 -471.333,E2 -471.333} C_VEL
LIN {X 0,Y 608.506,Z 323.474,A -85,B 0,C 180,E1 -472.315,E2 -472.315} C_VEL
LIN {X 0,Y 608.458,Z 323.317,A -85,B 0,C 180,E1 -474.572,E2 -474.572} C_VEL
LIN {X 0,Y 608.476,Z 323.31,A -85,B 0,C 180,E1 -477.207,E2 -477.207} C_VEL
LIN {X 0,Y 608.476,Z 323.317,A -85,B 0,C 180,E1 -479.973,E2 -479.973} C_VEL
LIN {X 0,Y 608.455,Z 323.313,A -85,B 0,C 180,E1 -482.88,E2 -482.88} C_VEL
LIN {X 0,Y 608.447,Z 323.314,A -85,B 0,C 180,E1 -485.278,E2 -485.278} C_VEL
LIN {X 0,Y 608.472,Z 323.316,A -85,B 0,C 180,E1 -488.241,E2 -488.241} C_VEL
LIN {X 0,Y 608.457,Z 323.314,A -85,B 0,C 180,E1 -491.342,E2 -491.342} C_VEL
LIN {X 0,Y 608.456,Z 323.316,A -85,B 0,C 180,E1 -494.264,E2 -494.264} C_VEL
LIN {X 0,Y 608.453,Z 323.313,A -85,B 0,C 180,E1 -497.04,E2 -497.04} C_VEL
LIN {X 0,Y 608.457,Z 323.321,A -85,B 0,C 180,E1 -499.697,E2 -499.697} C_VEL
LIN {X 0,Y 608.47,Z 323.313,A -85,B 0,C 180,E1 -502.254,E2 -502.254} C_VEL
LIN {X 0,Y 608.443,Z 323.315,A -85,B 0,C 180,E1 -505.096,E2 -505.096} C_VEL
LIN {X 0,Y 608.471,Z 323.316,A -85,B 0,C 180,E1 -507.906,E2 -507.906} C_VEL
LIN {X 0,Y 608.463,Z 323.313,A -85,B 0,C 180,E1 -510.22,E2 -510.22} C_VEL
LIN {X 0,Y 608.479,Z 323.31,A -85,B 0,C 180,E1 -512.793,E2 -512.793} C_VEL
LIN {X 0,Y 608.485,Z 323.51,A -85,B 0,C 180,E1 -515.461,E2 -515.461} C_VEL
LIN {X 0,Y 608.654,Z 332.048,A -85,B 0,C 180,E1 -516.524,E2 -516.524} C_VEL
LIN {X 0,Y 608.601,Z 356.517,A -85,B 0,C 180,E1 -519.466,E2 -519.466} C_VEL
LIN {X 0,Y 608.533,Z 380.985,A -85,B 0,C 180,E1 -522.352,E2 -522.352} C_VEL
LIN {X 0,Y 608.508,Z 404.713,A -85,B 0,C 180,E1 -525.109,E2 -525.109} C_VEL
LIN {X 0,Y 608.5,Z 421.137,A -85,B 0,C 180,E1 -526.984,E2 -526.984} C_VEL
LIN {X 0,Y 608.581,Z 424.216,A -85,B 0,C 180,E1 -527.05,E2 -527.05} C_VEL
LIN {X 0,Y 608.541,Z 530.292,A -85,B 0,C 180,E1 -528.319,E2 -528.319} C_VEL
LIN {X 0,Y 608.538,Z 543.622,A -85,B 0,C 180,E1 -528.614,E2 -528.614} C_VEL
LIN {X 0,Y 608.529,Z 556.856,A -85,B 0,C 180,E1 -529.055,E2 -529.055} C_VEL
LIN {X 0,Y 608.504,Z 568.871,A -85,B 0,C 180,E1 -529.603,E2 -529.603} C_VEL
LIN {X 0,Y 608.494,Z 580.291,A -85,B 0,C 180,E1 -530.275,E2 -530.275} C_VEL
LIN {X 0,Y 608.474,Z 590.585,A -85,B 0,C 180,E1 -531.029,E2 -531.029} C_VEL
LIN {X 0,Y 608.464,Z 599.851,A -85,B 0,C 180,E1 -531.866,E2 -531.866} C_VEL
LIN {X 0,Y 608.467,Z 608.824,A -85,B 0,C 180,E1 -532.867,E2 -532.867} C_VEL
LIN {X 0,Y 608.444,Z 616.056,A -85,B 0,C 180,E1 -533.867,E2 -533.867} C_VEL
LIN {X 0,Y 608.462,Z 620.935,A -85,B 0,C 180,E1 -534.698,E2 -534.698} C_VEL
LIN {X 0,Y 608.439,Z 625.679,A -85,B 0,C 180,E1 -535.694,E2 -535.694} C_VEL
LIN {X 0,Y 608.426,Z 629.312,A -85,B 0,C 180,E1 -536.689,E2 -536.689} C_VEL
LIN {X 0,Y 608.425,Z 631.191,A -85,B 0,C 180,E1 -537.352,E2 -537.352} C_VEL
LIN {X 0,Y 608.442,Z 632.627,A -85,B 0,C 180,E1 -538.014,E2 -538.014} C_VEL
LIN {X 0,Y 608.439,Z 634.252,A -85,B 0,C 180,E1 -539.338,E2 -539.338} C_VEL
LIN {X 0,Y 608.434,Z 634.495,A -85,B 0,C 180,E1 -540,E2 -540} C_VEL
LIN {X 0,Y 608.439,Z 634.315,A -85,B 0,C 180,E1 -540.662,E2 -540.662} C_VEL
LIN {X 0,Y 608.441,Z 632.776,A -85,B 0,C 180,E1 -541.986,E2 -541.986} C_VEL
LIN {X 0,Y 608.426,Z 631.418,A -85,B 0,C 180,E1 -542.648,E2 -542.648} C_VEL
LIN {X 0,Y 608.45,Z 628.542,A -85,B 0,C 180,E1 -543.642,E2 -543.642} C_VEL
LIN {X 0,Y 608.433,Z 624.643,A -85,B 0,C 180,E1 -544.638,E2 -544.638} C_VEL
LIN {X 0,Y 608.449,Z 619.612,A -85,B 0,C 180,E1 -545.634,E2 -545.634} C_VEL
LIN {X 0,Y 608.442,Z 613.294,A -85,B 0,C 180,E1 -546.633,E2 -546.633} C_VEL
LIN {X 0,Y 608.475,Z 605.379,A -85,B 0,C 180,E1 -547.633,E2 -547.633} C_VEL
LIN {X 0,Y 608.472,Z 595.535,A -85,B 0,C 180,E1 -548.636,E2 -548.636} C_VEL
LIN {X 0,Y 608.477,Z 593.429,A -85,B 0,C 180,E1 -548.82,E2 -548.82} C_VEL
LIN {X 0,Y 607.81,Z 589.094,A -85,B 0,C 180,E1 -549.19,E2 -549.19} C_VEL
LIN {X 0,Y 604.968,Z 581.845,A -85,B 0,C 180,E1 -549.77,E2 -549.77} C_VEL
LIN {X 0,Y 602.15,Z 574.199,A -85,B 0,C 180,E1 -550.302,E2 -550.302} C_VEL
LIN {X 0,Y 601.522,Z 569.142,A -85,B 0,C 180,E1 -550.595,E2 -550.595} C_VEL
LIN {X 0,Y 601.548,Z 556.654,A -85,B 0,C 180,E1 -551.172,E2 -551.172} C_VEL
LIN {X 0,Y 601.609,Z 543.809,A -85,B 0,C 180,E1 -551.604,E2 -551.604} C_VEL
LIN {X 0,Y 601.633,Z 530.569,A -85,B 0,C 180,E1 -551.903,E2 -551.903} C_VEL
LIN {X 0,Y 601.587,Z 422.114,A -85,B 0,C 180,E1 -553.222,E2 -553.222} C_VEL
LIN {X 0,Y 601.476,Z 420.721,A -85,B 0,C 180,E1 -553.3,E2 -553.3} C_VEL
LIN {X 0,Y 601.551,Z 398.069,A -85,B 0,C 180,E1 -555.935,E2 -555.935} C_VEL
LIN {X 0,Y 601.617,Z 374.227,A -85,B 0,C 180,E1 -558.751,E2 -558.751} C_VEL
LIN {X 0,Y 601.737,Z 350.589,A -85,B 0,C 180,E1 -561.587,E2 -561.587} C_VEL
LIN {X 0,Y 601.845,Z 326.594,A -85,B 0,C 180,E1 -564.522,E2 -564.522} C_VEL
LIN {X 0,Y 601.457,Z 324.321,A -85,B 0,C 180,E1 -564.855,E2 -564.855} C_VEL
LIN {X 0,Y 601.406,Z 324.192,A -85,B 0,C 180,E1 -567.868,E2 -567.868} C_VEL
LIN {X 0,Y 601.432,Z 324.193,A -85,B 0,C 180,E1 -570.164,E2 -570.164} C_VEL
LIN {X 0,Y 601.429,Z 324.193,A -85,B 0,C 180,E1 -572.716,E2 -572.716} C_VEL
LIN {X 0,Y 601.394,Z 324.193,A -85,B 0,C 180,E1 -575.111,E2 -575.111} C_VEL
LIN {X 0,Y 601.438,Z 324.186,A -85,B 0,C 180,E1 -577.419,E2 -577.419} C_VEL
LIN {X 0,Y 601.404,Z 324.196,A -85,B 0,C 180,E1 -579.996,E2 -579.996} C_VEL
LIN {X 0,Y 601.415,Z 324.192,A -85,B 0,C 180,E1 -582.67,E2 -582.67} C_VEL
LIN {X 0,Y 601.403,Z 324.191,A -85,B 0,C 180,E1 -585.479,E2 -585.479} C_VEL
LIN {X 0,Y 601.424,Z 324.194,A -85,B 0,C 180,E1 -588.407,E2 -588.407} C_VEL
LIN {X 0,Y 601.416,Z 324.189,A -85,B 0,C 180,E1 -590.873,E2 -590.873} C_VEL
LIN {X 0,Y 601.409,Z 324.191,A -85,B 0,C 180,E1 -593.417,E2 -593.417} C_VEL
LIN {X 0,Y 601.438,Z 324.196,A -85,B 0,C 180,E1 -596.064,E2 -596.064} C_VEL
LIN {X 0,Y 601.424,Z 324.19,A -85,B 0,C 180,E1 -598.545,E2 -598.545} C_VEL
LIN {X 0,Y 601.435,Z 324.188,A -85,B 0,C 180,E1 -601.373,E2 -601.373} C_VEL
LIN {X 0,Y 601.414,Z 324.195,A -85,B 0,C 180,E1 -604.133,E2 -604.133} C_VEL
LIN {X 0,Y 601.422,Z 324.192,A -85,B 0,C 180,E1 -606.589,E2 -606.589} C_VEL
LIN {X 0,Y 601.48,Z 324.364,A -85,B 0,C 180,E1 -607.58,E2 -607.58} C_VEL
LIN {X 0,Y 601.679,Z 330.142,A -85,B 0,C 180,E1 -608.411,E2 -608.411} C_VEL
LIN {X 0,Y 601.566,Z 351.929,A -85,B 0,C 180,E1 -611.377,E2 -611.377} C_VEL
LIN {X 0,Y 601.539,Z 372.155,A -85,B 0,C 180,E1 -614.064,E2 -614.064} C_VEL
LIN {X 0,Y 601.829,Z 375.429,A -85,B 0,C 180,E1 -614.137,E2 -614.137} C_VEL
LIN {X 0,Y 601.734,Z 508.892,A -85,B 0,C 180,E1 -615.767,E2 -615.767} C_VEL
LIN {X 0,Y 601.715,Z 522.907,A -85,B 0,C 180,E1 -616.063,E2 -616.063} C_VEL
LIN {X 0,Y 601.668,Z 537.638,A -85,B 0,C 180,E1 -616.532,E2 -616.532} C_VEL
LIN {X 0,Y 601.608,Z 550.675,A -85,B 0,C 180,E1 -617.089,E2 -617.089} C_VEL
LIN {X 0,Y 601.551,Z 563.336,A -85,B 0,C 180,E1 -617.774,E2 -617.774} C_VEL
LIN {X 0,Y 601.506,Z 574.855,A -85,B 0,C 180,E1 -618.542,E2 -618.542} C_VEL
LIN {X 0,Y 601.482,Z 585.416,A -85,B 0,C 180,E1 -619.395,E2 -619.395} C_VEL
LIN {X 0,Y 601.431,Z 595.898,A -85,B 0,C 180,E1 -620.414,E2 -620.414} C_VEL
LIN {X 0,Y 601.406,Z 604.54,A -85,B 0,C 180,E1 -621.43,E2 -621.43} C_VEL
LIN {X 0,Y 601.392,Z 612.838,A -85,B 0,C 180,E1 -622.613,E2 -622.613} C_VEL
LIN {X 0,Y 601.361,Z 618.513,A -85,B 0,C 180,E1 -623.605,E2 -623.605} C_VEL
LIN {X 0,Y 601.352,Z 623.378,A -85,B 0,C 180,E1 -624.634,E2 -624.634} C_VEL
LIN {X 0,Y 601.345,Z 628.3,A -85,B 0,C 180,E1 -625.978,E2 -625.978} C_VEL
LIN {X 0,Y 601.324,Z 631.731,A -85,B 0,C 180,E1 -627.32,E2 -627.32} C_VEL
LIN {X 0,Y 601.346,Z 633.773,A -85,B 0,C 180,E1 -628.66,E2 -628.66} C_VEL
LIN {X 0,Y 601.334,Z 634.495,A -85,B 0,C 180,E1 -629.999,E2 -629.999} C_VEL
LIN {X 0,Y 601.342,Z 633.879,A -85,B 0,C 180,E1 -631.339,E2 -631.339} C_VEL
LIN {X 0,Y 601.321,Z 631.926,A -85,B 0,C 180,E1 -632.679,E2 -632.679} C_VEL
LIN {X 0,Y 601.346,Z 628.589,A -85,B 0,C 180,E1 -634.02,E2 -634.02} C_VEL
LIN {X 0,Y 601.355,Z 623.766,A -85,B 0,C 180,E1 -635.364,E2 -635.364} C_VEL
LIN {X 0,Y 601.355,Z 617.299,A -85,B 0,C 180,E1 -636.711,E2 -636.711} C_VEL
LIN {X 0,Y 601.399,Z 610.096,A -85,B 0,C 180,E1 -637.891,E2 -637.891} C_VEL
LIN {X 0,Y 601.429,Z 601.203,A -85,B 0,C 180,E1 -639.076,E2 -639.076} C_VEL
LIN {X 0,Y 601.439,Z 591.866,A -85,B 0,C 180,E1 -640.094,E2 -640.094} C_VEL
LIN {X 0,Y 601.505,Z 581.247,A -85,B 0,C 180,E1 -641.05,E2 -641.05} C_VEL
LIN {X 0,Y 601.545,Z 570.11,A -85,B 0,C 180,E1 -641.882,E2 -641.882} C_VEL
LIN {X 0,Y 601.563,Z 557.49,A -85,B 0,C 180,E1 -642.653,E2 -642.653} C_VEL
LIN {X 0,Y 601.627,Z 545.222,A -85,B 0,C 180,E1 -643.252,E2 -643.252} C_VEL
LIN {X 0,Y 601.697,Z 531.167,A -85,B 0,C 180,E1 -643.782,E2 -643.782} C_VEL
LIN {X 0,Y 601.728,Z 517.512,A -85,B 0,C 180,E1 -644.154,E2 -644.154} C_VEL
LIN {X 0,Y 601.753,Z 503.64,A -85,B 0,C 180,E1 -644.4,E2 -644.4} C_VEL
LIN {X 0,Y 601.706,Z 373.292,A -85,B 0,C 180,E1 -645.985,E2 -645.985} C_VEL
LIN {X 0,Y 601.515,Z 371.726,A -85,B 0,C 180,E1 -646.066,E2 -646.066} C_VEL
LIN {X 0,Y 601.56,Z 350.858,A -85,B 0,C 180,E1 -648.858,E2 -648.858} C_VEL
LIN {X 0,Y 601.688,Z 329.501,A -85,B 0,C 180,E1 -651.767,E2 -651.767} C_VEL
LIN {X 0,Y 601.459,Z 324.411,A -85,B 0,C 180,E1 -652.5,E2 -652.5} C_VEL
LIN {X 0,Y 601.404,Z 324.193,A -85,B 0,C 180,E1 -654.877,E2 -654.877} C_VEL
LIN {X 0,Y 601.422,Z 324.193,A -85,B 0,C 180,E1 -657.866,E2 -657.866} C_VEL
LIN {X 0,Y 601.447,Z 324.195,A -85,B 0,C 180,E1 -660.162,E2 -660.162} C_VEL
LIN {X 0,Y 601.421,Z 324.19,A -85,B 0,C 180,E1 -662.715,E2 -662.715} C_VEL
LIN {X 0,Y 601.417,Z 324.189,A -85,B 0,C 180,E1 -665.114,E2 -665.114} C_VEL
LIN {X 0,Y 601.431,Z 324.189,A -85,B 0,C 180,E1 -667.418,E2 -667.418} C_VEL
LIN {X 0,Y 601.412,Z 324.199,A -85,B 0,C 180,E1 -669.993,E2 -669.993} C_VEL
LIN {X 0,Y 601.406,Z 324.191,A -85,B 0,C 180,E1 -672.669,E2 -672.669} C_VEL
LIN {X 0,Y 601.419,Z 324.192,A -85,B 0,C 180,E1 -675.481,E2 -675.481} C_VEL
LIN {X 0,Y 601.423,Z 324.19,A -85,B 0,C 180,E1 -678.405,E2 -678.405} C_VEL
LIN {X 0,Y 601.43,Z 324.187,A -85,B 0,C 180,E1 -680.875,E2 -680.875} C_VEL
LIN {X 0,Y 601.437,Z 324.197,A -85,B 0,C 180,E1 -683.733,E2 -683.733} C_VEL
LIN {X 0,Y 601.425,Z 324.188,A -85,B 0,C 180,E1 -686.686,E2 -686.686} C_VEL
LIN {X 0,Y 601.425,Z 324.19,A -85,B 0,C 180,E1 -689.058,E2 -689.058} C_VEL
LIN {X 0,Y 601.435,Z 324.192,A -85,B 0,C 180,E1 -691.373,E2 -691.373} C_VEL
LIN {X 0,Y 601.403,Z 324.199,A -85,B 0,C 180,E1 -693.636,E2 -693.636} C_VEL
LIN {X 0,Y 601.416,Z 324.189,A -85,B 0,C 180,E1 -696.589,E2 -696.589} C_VEL
LIN {X 0,Y 601.431,Z 324.197,A -85,B 0,C 180,E1 -699.478,E2 -699.478} C_VEL
LIN {X 0,Y 601.397,Z 324.191,A -85,B 0,C 180,E1 -702.312,E2 -702.312} C_VEL
LIN {X 0,Y 601.414,Z 324.189,A -85,B 0,C 180,E1 -704.409,E2 -704.409} C_VEL
LIN {X 0,Y 601.424,Z 324.197,A -85,B 0,C 180,E1 -707.172,E2 -707.172} C_VEL
LIN {X 0,Y 601.43,Z 324.188,A -85,B 0,C 180,E1 -709.905,E2 -709.905} C_VEL
LIN {X 0,Y 601.448,Z 324.187,A -85,B 0,C 180,E1 -712.615,E2 -712.615} C_VEL
LIN {X 0,Y 601.429,Z 324.194,A -85,B 0,C 180,E1 -715.308,E2 -715.308} C_VEL
LIN {X 0,Y 601.418,Z 324.188,A -85,B 0,C 180,E1 -717.991,E2 -717.991} C_VEL
LIN {X 0,Y 601.455,Z 324.189,A -85,B 0,C 180,E1 -720.669,E2 -720.669} C_VEL
LIN {X 0,Y 601.433,Z 324.19,A -85,B 0,C 180,E1 -723.349,E2 -723.349} C_VEL
LIN {X 0,Y 601.405,Z 324.191,A -85,B 0,C 180,E1 -726.037,E2 -726.037} C_VEL
LIN {X 0,Y 601.438,Z 324.195,A -85,B 0,C 180,E1 -728.738,E2 -728.738} C_VEL
LIN {X 0,Y 601.429,Z 324.188,A -85,B 0,C 180,E1 -731.458,E2 -731.458} C_VEL
LIN {X 0,Y 601.411,Z 324.192,A -85,B 0,C 180,E1 -734.206,E2 -734.206} C_VEL
LIN {X 0,Y 601.431,Z 324.193,A -85,B 0,C 180,E1 -736.986,E2 -736.986} C_VEL
LIN {X 0,Y 601.404,Z 324.191,A -85,B 0,C 180,E1 -739.809,E2 -739.809} C_VEL
LIN {X 0,Y 601.447,Z 324.194,A -85,B 0,C 180,E1 -742.682,E2 -742.682} C_VEL
LIN {X 0,Y 601.4,Z 324.196,A -85,B 0,C 180,E1 -744.879,E2 -744.879} C_VEL
LIN {X 0,Y 601.419,Z 324.189,A -85,B 0,C 180,E1 -747.867,E2 -747.867} C_VEL
LIN {X 0,Y 601.419,Z 324.193,A -85,B 0,C 180,E1 -750.165,E2 -750.165} C_VEL
LIN {X 0,Y 601.426,Z 324.193,A -85,B 0,C 180,E1 -752.718,E2 -752.718} C_VEL
LIN {X 0,Y 601.404,Z 324.191,A -85,B 0,C 180,E1 -755.115,E2 -755.115} C_VEL
LIN {X 0,Y 601.429,Z 324.186,A -85,B 0,C 180,E1 -757.42,E2 -757.42} C_VEL
LIN {X 0,Y 601.406,Z 324.196,A -85,B 0,C 180,E1 -759.995,E2 -759.995} C_VEL
LIN {X 0,Y 601.432,Z 324.19,A -85,B 0,C 180,E1 -762.669,E2 -762.669} C_VEL
LIN {X 0,Y 601.418,Z 324.189,A -85,B 0,C 180,E1 -765.483,E2 -765.483} C_VEL
LIN {X 0,Y 601.42,Z 324.194,A -85,B 0,C 180,E1 -768.407,E2 -768.407} C_VEL
LIN {X 0,Y 601.433,Z 324.187,A -85,B 0,C 180,E1 -770.877,E2 -770.877} C_VEL
LIN {X 0,Y 601.441,Z 324.192,A -85,B 0,C 180,E1 -773.734,E2 -773.734} C_VEL
LIN {X 0,Y 601.432,Z 324.195,A -85,B 0,C 180,E1 -776.065,E2 -776.065} C_VEL
LIN {X 0,Y 601.439,Z 324.188,A -85,B 0,C 180,E1 -778.543,E2 -778.543} C_VEL
LIN {X 0,Y 601.435,Z 324.188,A -85,B 0,C 180,E1 -781.375,E2 -781.375} C_VEL
LIN {X 0,Y 601.414,Z 324.195,A -85,B 0,C 180,E1 -784.133,E2 -784.133} C_VEL
LIN {X 0,Y 601.421,Z 324.192,A -85,B 0,C 180,E1 -786.591,E2 -786.591} C_VEL
LIN {X 0,Y 601.452,Z 324.445,A -85,B 0,C 180,E1 -787.553,E2 -787.553} C_VEL
LIN {X 0,Y 601.687,Z 329.174,A -85,B 0,C 180,E1 -788.233,E2 -788.233} C_VEL
LIN {X 0,Y 601.561,Z 350.521,A -85,B 0,C 180,E1 -791.141,E2 -791.141} C_VEL
LIN {X 0,Y 601.521,Z 371.019,A -85,B 0,C 180,E1 -793.891,E2 -793.891} C_VEL
LIN {X 0,Y 601.6,Z 372.676,A -85,B 0,C 180,E1 -794.045,E2 -794.045} C_VEL
LIN {X 0,Y 601.82,Z 379.277,A -85,B 0,C 180,E1 -794.138,E2 -794.138} C_VEL
LIN {X 0,Y 601.754,Z 508.969,A -85,B 0,C 180,E1 -795.722,E2 -795.722} C_VEL
LIN {X 0,Y 601.72,Z 523.275,A -85,B 0,C 180,E1 -796.029,E2 -796.029} C_VEL
LIN {X 0,Y 601.659,Z 535.939,A -85,B 0,C 180,E1 -796.422,E2 -796.422} C_VEL
LIN {X 0,Y 601.63,Z 548.115,A -85,B 0,C 180,E1 -796.92,E2 -796.92} C_VEL
LIN {X 0,Y 601.575,Z 561.282,A -85,B 0,C 180,E1 -797.605,E2 -797.605} C_VEL
LIN {X 0,Y 601.51,Z 573.163,A -85,B 0,C 180,E1 -798.373,E2 -798.373} C_VEL
LIN {X 0,Y 601.489,Z 584.004,A -85,B 0,C 180,E1 -799.226,E2 -799.226} C_VEL
LIN {X 0,Y 601.422,Z 594.717,A -85,B 0,C 180,E1 -800.246,E2 -800.246} C_VEL
LIN {X 0,Y 601.406,Z 603.565,A -85,B 0,C 180,E1 -801.263,E2 -801.263} C_VEL
LIN {X 0,Y 601.406,Z 612.045,A -85,B 0,C 180,E1 -802.447,E2 -802.447} C_VEL
LIN {X 0,Y 601.361,Z 618.752,A -85,B 0,C 180,E1 -803.605,E2 -803.605} C_VEL
LIN {X 0,Y 601.355,Z 623.571,A -85,B 0,C 180,E1 -804.636,E2 -804.636} C_VEL
LIN {X 0,Y 601.343,Z 628.445,A -85,B 0,C 180,E1 -805.98,E2 -805.98} C_VEL
LIN {X 0,Y 601.324,Z 631.833,A -85,B 0,C 180,E1 -807.321,E2 -807.321} C_VEL
LIN {X 0,Y 601.342,Z 633.832,A -85,B 0,C 180,E1 -808.661,E2 -808.661} C_VEL
LIN {X 0,Y 601.333,Z 634.5,A -85,B 0,C 180,E1 -810.001,E2 -810.001} C_VEL
LIN {X 0,Y 601.342,Z 633.83,A -85,B 0,C 180,E1 -811.34,E2 -811.34} C_VEL
LIN {X 0,Y 601.324,Z 631.829,A -85,B 0,C 180,E1 -812.68,E2 -812.68} C_VEL
LIN {X 0,Y 601.343,Z 628.439,A -85,B 0,C 180,E1 -814.022,E2 -814.022} C_VEL
LIN {X 0,Y 601.355,Z 623.564,A -85,B 0,C 180,E1 -815.366,E2 -815.366} C_VEL
LIN {X 0,Y 601.356,Z 617.047,A -85,B 0,C 180,E1 -816.712,E2 -816.712} C_VEL
LIN {X 0,Y 601.398,Z 609.793,A -85,B 0,C 180,E1 -817.893,E2 -817.893} C_VEL
LIN {X 0,Y 601.43,Z 600.816,A -85,B 0,C 180,E1 -819.077,E2 -819.077} C_VEL
LIN {X 0,Y 601.44,Z 591.383,A -85,B 0,C 180,E1 -820.096,E2 -820.096} C_VEL
LIN {X 0,Y 601.505,Z 580.69,A -85,B 0,C 180,E1 -821.051,E2 -821.051} C_VEL
LIN {X 0,Y 601.544,Z 569.415,A -85,B 0,C 180,E1 -821.884,E2 -821.884} C_VEL
LIN {X 0,Y 601.564,Z 556.629,A -85,B 0,C 180,E1 -822.654,E2 -822.654} C_VEL
LIN {X 0,Y 601.633,Z 544.142,A -85,B 0,C 180,E1 -823.254,E2 -823.254} C_VEL
LIN {X 0,Y 601.694,Z 530.815,A -85,B 0,C 180,E1 -823.749,E2 -823.749} C_VEL
LIN {X 0,Y 601.736,Z 516.48,A -85,B 0,C 180,E1 -824.135,E2 -824.135} C_VEL
LIN {X 0,Y 601.753,Z 502.029,A -85,B 0,C 180,E1 -824.377,E2 -824.377} C_VEL
LIN {X 0,Y 601.685,Z 373.261,A -85,B 0,C 180,E1 -825.941,E2 -825.941} C_VEL
LIN {X 0,Y 601.505,Z 371.699,A -85,B 0,C 180,E1 -826.024,E2 -826.024} C_VEL
LIN {X 0,Y 601.565,Z 352.262,A -85,B 0,C 180,E1 -828.623,E2 -828.623} C_VEL
LIN {X 0,Y 601.678,Z 330.469,A -85,B 0,C 180,E1 -831.589,E2 -831.589} C_VEL
LIN {X 0,Y 601.487,Z 324.594,A -85,B 0,C 180,E1 -832.42,E2 -832.42} C_VEL
LIN {X 0,Y 601.416,Z 324.196,A -85,B 0,C 180,E1 -832.684,E2 -832.684} C_VEL
LIN {X 0,Y 601.405,Z 324.192,A -85,B 0,C 180,E1 -834.879,E2 -834.879} C_VEL
LIN {X 0,Y 601.424,Z 324.194,A -85,B 0,C 180,E1 -837.868,E2 -837.868} C_VEL
LIN {X 0,Y 601.434,Z 324.197,A -85,B 0,C 180,E1 -840.164,E2 -840.164} C_VEL
LIN {X 0,Y 601.423,Z 324.19,A -85,B 0,C 180,E1 -842.715,E2 -842.715} C_VEL
LIN {X 0,Y 601.418,Z 324.189,A -85,B 0,C 180,E1 -845.115,E2 -845.115} C_VEL
LIN {X 0,Y 601.438,Z 324.188,A -85,B 0,C 180,E1 -847.42,E2 -847.42} C_VEL
LIN {X 0,Y 601.407,Z 324.2,A -85,B 0,C 180,E1 -849.996,E2 -849.996} C_VEL
LIN {X 0,Y 601.411,Z 324.19,A -85,B 0,C 180,E1 -852.671,E2 -852.671} C_VEL
LIN {X 0,Y 601.431,Z 324.191,A -85,B 0,C 180,E1 -855.482,E2 -855.482} C_VEL
LIN {X 0,Y 601.427,Z 324.19,A -85,B 0,C 180,E1 -858.407,E2 -858.407} C_VEL
LIN {X 0,Y 601.433,Z 324.194,A -85,B 0,C 180,E1 -861.53,E2 -861.53} C_VEL
LIN {X 0,Y 601.388,Z 324.195,A -85,B 0,C 180,E1 -864.245,E2 -864.245} C_VEL
LIN {X 0,Y 601.422,Z 324.189,A -85,B 0,C 180,E1 -866.686,E2 -866.686} C_VEL
LIN {X 0,Y 601.416,Z 324.191,A -85,B 0,C 180,E1 -869.058,E2 -869.058} C_VEL
LIN {X 0,Y 601.437,Z 324.194,A -85,B 0,C 180,E1 -871.373,E2 -871.373} C_VEL
LIN {X 0,Y 601.405,Z 324.201,A -85,B 0,C 180,E1 -873.636,E2 -873.636} C_VEL
LIN {X 0,Y 601.462,Z 324.381,A -85,B 0,C 180,E1 -875.258,E2 -875.258} C_VEL
LIN {X 0,Y 601.826,Z 328.077,A -85,B 0,C 180,E1 -875.75,E2 -875.75} C_VEL
LIN {X 0,Y 601.735,Z 349.848,A -85,B 0,C 180,E1 -878.413,E2 -878.413} C_VEL
LIN {X 0,Y 601.628,Z 374.473,A -85,B 0,C 180,E1 -881.369,E2 -881.369} C_VEL
LIN {X 0,Y 601.542,Z 400.268,A -85,B 0,C 180,E1 -884.412,E2 -884.412} C_VEL
LIN {X 0,Y 601.499,Z 421.143,A -85,B 0,C 180,E1 -886.83,E2 -886.83} C_VEL
LIN {X 0,Y 601.679,Z 424.262,A -85,B 0,C 180,E1 -886.898,E2 -886.898} C_VEL
LIN {X 0,Y 601.616,Z 530.311,A -85,B 0,C 180,E1 -888.182,E2 -888.182} C_VEL
LIN {X 0,Y 601.59,Z 543.65,A -85,B 0,C 180,E1 -888.481,E2 -888.481} C_VEL
LIN {X 0,Y 601.567,Z 556.728,A -85,B 0,C 180,E1 -888.921,E2 -888.921} C_VEL
LIN {X 0,Y 601.513,Z 568.886,A -85,B 0,C 180,E1 -889.481,E2 -889.481} C_VEL
LIN {X 0,Y 601.459,Z 580.303,A -85,B 0,C 180,E1 -890.16,E2 -890.16} C_VEL
LIN {X 0,Y 601.438,Z 590.594,A -85,B 0,C 180,E1 -890.924,E2 -890.924} C_VEL
LIN {X 0,Y 601.411,Z 599.859,A -85,B 0,C 180,E1 -891.77,E2 -891.77} C_VEL
LIN {X 0,Y 601.389,Z 608.831,A -85,B 0,C 180,E1 -892.783,E2 -892.783} C_VEL
LIN {X 0,Y 601.376,Z 615.97,A -85,B 0,C 180,E1 -893.781,E2 -893.781} C_VEL
LIN {X 0,Y 601.373,Z 620.94,A -85,B 0,C 180,E1 -894.635,E2 -894.635} C_VEL
LIN {X 0,Y 601.353,Z 625.682,A -85,B 0,C 180,E1 -895.643,E2 -895.643} C_VEL
LIN {X 0,Y 601.345,Z 629.315,A -85,B 0,C 180,E1 -896.65,E2 -896.65} C_VEL
LIN {X 0,Y 601.324,Z 631.192,A -85,B 0,C 180,E1 -897.32,E2 -897.32} C_VEL
LIN {X 0,Y 601.341,Z 632.627,A -85,B 0,C 180,E1 -897.991,E2 -897.991} C_VEL
LIN {X 0,Y 601.339,Z 634.252,A -85,B 0,C 180,E1 -899.33,E2 -899.33} C_VEL
LIN {X 0,Y 601.335,Z 634.496,A -85,B 0,C 180,E1 -900,E2 -900} C_VEL
LIN {X 0,Y 601.339,Z 634.315,A -85,B 0,C 180,E1 -900.67,E2 -900.67} C_VEL
LIN {X 0,Y 601.34,Z 632.775,A -85,B 0,C 180,E1 -902.009,E2 -902.009} C_VEL
LIN {X 0,Y 601.326,Z 631.417,A -85,B 0,C 180,E1 -902.68,E2 -902.68} C_VEL
LIN {X 0,Y 601.368,Z 628.541,A -85,B 0,C 180,E1 -903.685,E2 -903.685} C_VEL
LIN {X 0,Y 601.337,Z 624.642,A -85,B 0,C 180,E1 -904.693,E2 -904.693} C_VEL
LIN {X 0,Y 601.373,Z 619.611,A -85,B 0,C 180,E1 -905.701,E2 -905.701} C_VEL
LIN {X 0,Y 601.383,Z 613.289,A -85,B 0,C 180,E1 -906.711,E2 -906.711} C_VEL
LIN {X 0,Y 601.396,Z 605.377,A -85,B 0,C 180,E1 -907.723,E2 -907.723} C_VEL
LIN {X 0,Y 601.437,Z 595.529,A -85,B 0,C 180,E1 -908.738,E2 -908.738} C_VEL
LIN {X 0,Y 601.444,Z 585.209,A -85,B 0,C 180,E1 -909.585,E2 -909.585} C_VEL
LIN {X 0,Y 601.493,Z 573.596,A -85,B 0,C 180,E1 -910.349,E2 -910.349} C_VEL
LIN {X 0,Y 601.522,Z 569.142,A -85,B 0,C 180,E1 -910.595,E2 -910.595} C_VEL
LIN {X 0,Y 600.922,Z 564.014,A -85,B 0,C 180,E1 -910.868,E2 -910.868} C_VEL
LIN {X 0,Y 598.201,Z 555.55,A -85,B 0,C 180,E1 -911.286,E2 -911.286} C_VEL
LIN {X 0,Y 595.392,Z 546.798,A -85,B 0,C 180,E1 -911.641,E2 -911.641} C_VEL
LIN {X 0,Y 594.652,Z 541.22,A -85,B 0,C 180,E1 -911.814,E2 -911.814} C_VEL
LIN {X 0,Y 594.686,Z 527.769,A -85,B 0,C 180,E1 -912.087,E2 -912.087} C_VEL
LIN {X 0,Y 594.649,Z 422.758,A -85,B 0,C 180,E1 -913.368,E2 -913.368} C_VEL
LIN {X 0,Y 594.477,Z 420.92,A -85,B 0,C 180,E1 -913.437,E2 -913.437} C_VEL
LIN {X 0,Y 594.569,Z 396.58,A -85,B 0,C 180,E1 -916.304,E2 -916.304} C_VEL
LIN {X 0,Y 594.682,Z 373.156,A -85,B 0,C 180,E1 -919.107,E2 -919.107} C_VEL
LIN {X 0,Y 594.852,Z 350.584,A -85,B 0,C 180,E1 -921.849,E2 -921.849} C_VEL
LIN {X 0,Y 594.986,Z 328.701,A -85,B 0,C 180,E1 -924.559,E2 -924.559} C_VEL
LIN {X 0,Y 594.401,Z 325.215,A -85,B 0,C 180,E1 -925.055,E2 -925.055} C_VEL
LIN {X 0,Y 594.373,Z 325.068,A -85,B 0,C 180,E1 -927.523,E2 -927.523} C_VEL
LIN {X 0,Y 594.39,Z 325.073,A -85,B 0,C 180,E1 -930.328,E2 -930.328} C_VEL
LIN {X 0,Y 594.383,Z 325.068,A -85,B 0,C 180,E1 -932.95,E2 -932.95} C_VEL
LIN {X 0,Y 594.353,Z 325.069,A -85,B 0,C 180,E1 -935.409,E2 -935.409} C_VEL
LIN {X 0,Y 594.388,Z 325.069,A -85,B 0,C 180,E1 -937.941,E2 -937.941} C_VEL
LIN {X 0,Y 594.378,Z 325.068,A -85,B 0,C 180,E1 -940.821,E2 -940.821} C_VEL
LIN {X 0,Y 594.372,Z 325.066,A -85,B 0,C 180,E1 -943.299,E2 -943.299} C_VEL
LIN {X 0,Y 594.365,Z 325.076,A -85,B 0,C 180,E1 -946.161,E2 -946.161} C_VEL
LIN {X 0,Y 594.381,Z 325.069,A -85,B 0,C 180,E1 -948.535,E2 -948.535} C_VEL
LIN {X 0,Y 594.387,Z 325.065,A -85,B 0,C 180,E1 -951.296,E2 -951.296} C_VEL
LIN {X 0,Y 594.366,Z 325.073,A -85,B 0,C 180,E1 -953.756,E2 -953.756} C_VEL
LIN {X 0,Y 594.381,Z 325.071,A -85,B 0,C 180,E1 -956.238,E2 -956.238} C_VEL
LIN {X 0,Y 594.375,Z 325.068,A -85,B 0,C 180,E1 -958.649,E2 -958.649} C_VEL
LIN {X 0,Y 594.388,Z 325.063,A -85,B 0,C 180,E1 -961.042,E2 -961.042} C_VEL
LIN {X 0,Y 594.389,Z 325.072,A -85,B 0,C 180,E1 -963.977,E2 -963.977} C_VEL
LIN {X 0,Y 594.394,Z 325.071,A -85,B 0,C 180,E1 -966.295,E2 -966.295} C_VEL
LIN {X 0,Y 594.415,Z 325.267,A -85,B 0,C 180,E1 -967.428,E2 -967.428} C_VEL
LIN {X 0,Y 594.769,Z 328.839,A -85,B 0,C 180,E1 -967.965,E2 -967.965} C_VEL
LIN {X 0,Y 594.648,Z 348.448,A -85,B 0,C 180,E1 -970.674,E2 -970.674} C_VEL
LIN {X 0,Y 594.542,Z 369.365,A -85,B 0,C 180,E1 -973.518,E2 -973.518} C_VEL
LIN {X 0,Y 594.552,Z 372.17,A -85,B 0,C 180,E1 -973.871,E2 -973.871} C_VEL
LIN {X 0,Y 595.018,Z 375.475,A -85,B 0,C 180,E1 -973.95,E2 -973.95} C_VEL
LIN {X 0,Y 594.867,Z 509.709,A -85,B 0,C 180,E1 -975.612,E2 -975.612} C_VEL
LIN {X 0,Y 594.833,Z 523.716,A -85,B 0,C 180,E1 -975.921,E2 -975.921} C_VEL
LIN {X 0,Y 594.755,Z 537.653,A -85,B 0,C 180,E1 -976.373,E2 -976.373} C_VEL
LIN {X 0,Y 594.657,Z 550.674,A -85,B 0,C 180,E1 -976.936,E2 -976.936} C_VEL
LIN {X 0,Y 594.602,Z 561.922,A -85,B 0,C 180,E1 -977.542,E2 -977.542} C_VEL
LIN {X 0,Y 594.508,Z 573.706,A -85,B 0,C 180,E1 -978.319,E2 -978.319} C_VEL
LIN {X 0,Y 594.474,Z 585.427,A -85,B 0,C 180,E1 -979.268,E2 -979.268} C_VEL
LIN {X 0,Y 594.392,Z 595.897,A -85,B 0,C 180,E1 -980.299,E2 -980.299} C_VEL
LIN {X 0,Y 594.355,Z 604.535,A -85,B 0,C 180,E1 -981.328,E2 -981.328} C_VEL
LIN {X 0,Y 594.315,Z 612.841,A -85,B 0,C 180,E1 -982.525,E2 -982.525} C_VEL
LIN {X 0,Y 594.271,Z 619.005,A -85,B 0,C 180,E1 -983.62,E2 -983.62} C_VEL
LIN {X 0,Y 594.246,Z 624.778,A -85,B 0,C 180,E1 -984.91,E2 -984.91} C_VEL
LIN {X 0,Y 594.261,Z 628.304,A -85,B 0,C 180,E1 -985.93,E2 -985.93} C_VEL
LIN {X 0,Y 594.224,Z 631.731,A -85,B 0,C 180,E1 -987.288,E2 -987.288} C_VEL
LIN {X 0,Y 594.245,Z 633.77,A -85,B 0,C 180,E1 -988.644,E2 -988.644} C_VEL
LIN {X 0,Y 594.235,Z 634.495,A -85,B 0,C 180,E1 -989.999,E2 -989.999} C_VEL
LIN {X 0,Y 594.242,Z 633.875,A -85,B 0,C 180,E1 -991.355,E2 -991.355} C_VEL
LIN {X 0,Y 594.221,Z 631.917,A -85,B 0,C 180,E1 -992.711,E2 -992.711} C_VEL
LIN {X 0,Y 594.262,Z 628.589,A -85,B 0,C 180,E1 -994.068,E2 -994.068} C_VEL
LIN {X 0,Y 594.275,Z 623.766,A -85,B 0,C 180,E1 -995.428,E2 -995.428} C_VEL
LIN {X 0,Y 594.277,Z 617.298,A -85,B 0,C 180,E1 -996.791,E2 -996.791} C_VEL
LIN {X 0,Y 594.329,Z 610.087,A -85,B 0,C 180,E1 -997.986,E2 -997.986} C_VEL
LIN {X 0,Y 594.384,Z 601.197,A -85,B 0,C 180,E1 -999.184,E2 -999.184} C_VEL
LIN {X 0,Y 594.411,Z 591.858,A -85,B 0,C 180,E1 -1000.215,E2 -1000.215} C_VEL
LIN {X 0,Y 594.507,Z 581.863,A -85,B 0,C 180,E1 -1001.13,E2 -1001.13} C_VEL
LIN {X 0,Y 594.57,Z 571.351,A -85,B 0,C 180,E1 -1001.937,E2 -1001.937} C_VEL
LIN {X 0,Y 594.615,Z 560.546,A -85,B 0,C 180,E1 -1002.629,E2 -1002.629} C_VEL
LIN {X 0,Y 594.691,Z 547.186,A -85,B 0,C 180,E1 -1003.322,E2 -1003.322} C_VEL
LIN {X 0,Y 594.787,Z 533.541,A -85,B 0,C 180,E1 -1003.865,E2 -1003.865} C_VEL
LIN {X 0,Y 594.814,Z 519.842,A -85,B 0,C 180,E1 -1004.266,E2 -1004.266} C_VEL
LIN {X 0,Y 594.88,Z 505.787,A -85,B 0,C 180,E1 -1004.539,E2 -1004.539} C_VEL
LIN {X 0,Y 594.927,Z 374.436,A -85,B 0,C 180,E1 -1006.155,E2 -1006.155} C_VEL
LIN {X 0,Y 594.572,Z 372.215,A -85,B 0,C 180,E1 -1006.215,E2 -1006.215} C_VEL
LIN {X 0,Y 594.602,Z 352.397,A -85,B 0,C 180,E1 -1008.876,E2 -1008.876} C_VEL
LIN {X 0,Y 594.771,Z 332.113,A -85,B 0,C 180,E1 -1011.669,E2 -1011.669} C_VEL
LIN {X 0,Y 594.567,Z 326.127,A -85,B 0,C 180,E1 -1012.513,E2 -1012.513} C_VEL
LIN {X 0,Y 594.378,Z 325.141,A -85,B 0,C 180,E1 -1012.738,E2 -1012.738} C_VEL
LIN {X 0,Y 594.376,Z 325.067,A -85,B 0,C 180,E1 -1015.192,E2 -1015.192} C_VEL
LIN {X 0,Y 594.383,Z 325.067,A -85,B 0,C 180,E1 -1017.526,E2 -1017.526} C_VEL
LIN {X 0,Y 594.4,Z 325.071,A -85,B 0,C 180,E1 -1020.33,E2 -1020.33} C_VEL
LIN {X 0,Y 594.376,Z 325.066,A -85,B 0,C 180,E1 -1022.949,E2 -1022.949} C_VEL
LIN {X 0,Y 594.382,Z 325.067,A -85,B 0,C 180,E1 -1025.405,E2 -1025.405} C_VEL
LIN {X 0,Y 594.387,Z 325.074,A -85,B 0,C 180,E1 -1027.939,E2 -1027.939} C_VEL
LIN {X 0,Y 594.384,Z 325.065,A -85,B 0,C 180,E1 -1030.822,E2 -1030.822} C_VEL
LIN {X 0,Y 594.377,Z 325.076,A -85,B 0,C 180,E1 -1033.84,E2 -1033.84} C_VEL
LIN {X 0,Y 594.38,Z 325.065,A -85,B 0,C 180,E1 -1036.702,E2 -1036.702} C_VEL
LIN {X 0,Y 594.383,Z 325.07,A -85,B 0,C 180,E1 -1039.434,E2 -1039.434} C_VEL
LIN {X 0,Y 594.385,Z 325.064,A -85,B 0,C 180,E1 -1042.39,E2 -1042.39} C_VEL
LIN {X 0,Y 594.375,Z 325.066,A -85,B 0,C 180,E1 -1044.671,E2 -1044.671} C_VEL
LIN {X 0,Y 594.374,Z 325.069,A -85,B 0,C 180,E1 -1047.087,E2 -1047.087} C_VEL
LIN {X 0,Y 594.392,Z 325.071,A -85,B 0,C 180,E1 -1049.668,E2 -1049.668} C_VEL
LIN {X 0,Y 594.382,Z 325.064,A -85,B 0,C 180,E1 -1052.539,E2 -1052.539} C_VEL
LIN {X 0,Y 594.371,Z 325.067,A -85,B 0,C 180,E1 -1054.807,E2 -1054.807} C_VEL
LIN {X 0,Y 594.395,Z 325.071,A -85,B 0,C 180,E1 -1057.254,E2 -1057.254} C_VEL
LIN {X 0,Y 594.374,Z 325.068,A -85,B 0,C 180,E1 -1059.946,E2 -1059.946} C_VEL
LIN {X 0,Y 594.387,Z 325.067,A -85,B 0,C 180,E1 -1062.806,E2 -1062.806} C_VEL
LIN {X 0,Y 594.379,Z 325.068,A -85,B 0,C 180,E1 -1065.825,E2 -1065.825} C_VEL
LIN {X 0,Y 594.387,Z 325.065,A -85,B 0,C 180,E1 -1068.404,E2 -1068.404} C_VEL
LIN {X 0,Y 594.398,Z 325.072,A -85,B 0,C 180,E1 -1071.158,E2 -1071.158} C_VEL
LIN {X 0,Y 594.398,Z 325.071,A -85,B 0,C 180,E1 -1073.299,E2 -1073.299} C_VEL
LIN {X 0,Y 594.355,Z 325.068,A -85,B 0,C 180,E1 -1075.932,E2 -1075.932} C_VEL
LIN {X 0,Y 594.389,Z 325.064,A -85,B 0,C 180,E1 -1077.967,E2 -1077.967} C_VEL
LIN {X 0,Y 594.425,Z 325.065,A -85,B 0,C 180,E1 -1080.677,E2 -1080.677} C_VEL
LIN {X 0,Y 594.383,Z 325.068,A -85,B 0,C 180,E1 -1083.389,E2 -1083.389} C_VEL
LIN {X 0,Y 594.361,Z 325.068,A -85,B 0,C 180,E1 -1086.109,E2 -1086.109} C_VEL
LIN {X 0,Y 594.411,Z 325.062,A -85,B 0,C 180,E1 -1088.157,E2 -1088.157} C_VEL
LIN {X 0,Y 594.39,Z 325.07,A -85,B 0,C 180,E1 -1091.081,E2 -1091.081} C_VEL
LIN {X 0,Y 594.377,Z 325.066,A -85,B 0,C 180,E1 -1093.679,E2 -1093.679} C_VEL
LIN {X 0,Y 594.394,Z 325.074,A -85,B 0,C 180,E1 -1096.724,E2 -1096.724} C_VEL
LIN {X 0,Y 594.364,Z 325.068,A -85,B 0,C 180,E1 -1099.335,E2 -1099.335} C_VEL
LIN {X 0,Y 594.365,Z 325.067,A -85,B 0,C 180,E1 -1101.503,E2 -1101.503} C_VEL
LIN {X 0,Y 594.385,Z 325.065,A -85,B 0,C 180,E1 -1103.704,E2 -1103.704} C_VEL
LIN {X 0,Y 594.382,Z 325.071,A -85,B 0,C 180,E1 -1106.7,E2 -1106.7} C_VEL
LIN {X 0,Y 594.378,Z 325.065,A -85,B 0,C 180,E1 -1108.999,E2 -1108.999} C_VEL
LIN {X 0,Y 594.387,Z 325.064,A -85,B 0,C 180,E1 -1111.647,E2 -1111.647} C_VEL
LIN {X 0,Y 594.387,Z 325.071,A -85,B 0,C 180,E1 -1114.58,E2 -1114.58} C_VEL
LIN {X 0,Y 594.379,Z 325.064,A -85,B 0,C 180,E1 -1117.087,E2 -1117.087} C_VEL
LIN {X 0,Y 594.369,Z 325.069,A -85,B 0,C 180,E1 -1119.775,E2 -1119.775} C_VEL
LIN {X 0,Y 594.382,Z 325.073,A -85,B 0,C 180,E1 -1122.374,E2 -1122.374} C_VEL
LIN {X 0,Y 594.356,Z 325.067,A -85,B 0,C 180,E1 -1125.192,E2 -1125.192} C_VEL
LIN {X 0,Y 594.364,Z 325.07,A -85,B 0,C 180,E1 -1127.626,E2 -1127.626} C_VEL
LIN {X 0,Y 594.39,Z 325.07,A -85,B 0,C 180,E1 -1130.322,E2 -1130.322} C_VEL
LIN {X 0,Y 594.382,Z 325.065,A -85,B 0,C 180,E1 -1132.915,E2 -1132.915} C_VEL
LIN {X 0,Y 594.385,Z 325.074,A -85,B 0,C 180,E1 -1135.861,E2 -1135.861} C_VEL
LIN {X 0,Y 594.389,Z 325.066,A -85,B 0,C 180,E1 -1138.652,E2 -1138.652} C_VEL
LIN {X 0,Y 594.384,Z 325.063,A -85,B 0,C 180,E1 -1141.042,E2 -1141.042} C_VEL
LIN {X 0,Y 594.388,Z 325.071,A -85,B 0,C 180,E1 -1143.977,E2 -1143.977} C_VEL
LIN {X 0,Y 594.392,Z 325.071,A -85,B 0,C 180,E1 -1146.297,E2 -1146.297} C_VEL
LIN {X 0,Y 594.408,Z 325.245,A -85,B 0,C 180,E1 -1147.377,E2 -1147.377} C_VEL
LIN {X 0,Y 594.778,Z 329.174,A -85,B 0,C 180,E1 -1147.967,E2 -1147.967} C_VEL
LIN {X 0,Y 594.636,Z 350.428,A -85,B 0,C 180,E1 -1150.901,E2 -1150.901} C_VEL
LIN {X 0,Y 594.544,Z 371.935,A -85,B 0,C 180,E1 -1153.807,E2 -1153.807} C_VEL
LIN {X 0,Y 594.813,Z 373.911,A -85,B 0,C 180,E1 -1153.88,E2 -1153.88} C_VEL
LIN {X 0,Y 594.977,Z 393.586,A -85,B 0,C 180,E1 -1154.127,E2 -1154.127} C_VEL
LIN {X 0,Y 594.856,Z 509.937,A -85,B 0,C 180,E1 -1155.57,E2 -1155.57} C_VEL
LIN {X 0,Y 594.818,Z 524.169,A -85,B 0,C 180,E1 -1155.889,E2 -1155.889} C_VEL
LIN {X 0,Y 594.729,Z 537.737,A -85,B 0,C 180,E1 -1156.33,E2 -1156.33} C_VEL
LIN {X 0,Y 594.655,Z 551.657,A -85,B 0,C 180,E1 -1156.938,E2 -1156.938} C_VEL
LIN {X 0,Y 594.594,Z 564.112,A -85,B 0,C 180,E1 -1157.63,E2 -1157.63} C_VEL
LIN {X 0,Y 594.523,Z 576.57,A -85,B 0,C 180,E1 -1158.488,E2 -1158.488} C_VEL
LIN {X 0,Y 594.448,Z 587.846,A -85,B 0,C 180,E1 -1159.442,E2 -1159.442} C_VEL
LIN {X 0,Y 594.367,Z 597.858,A -85,B 0,C 180,E1 -1160.472,E2 -1160.472} C_VEL
LIN {X 0,Y 594.323,Z 606.177,A -85,B 0,C 180,E1 -1161.501,E2 -1161.501} C_VEL
LIN {X 0,Y 594.302,Z 614.131,A -85,B 0,C 180,E1 -1162.697,E2 -1162.697} C_VEL
LIN {X 0,Y 594.279,Z 620.531,A -85,B 0,C 180,E1 -1163.891,E2 -1163.891} C_VEL
LIN {X 0,Y 594.237,Z 626.202,A -85,B 0,C 180,E1 -1165.252,E2 -1165.252} C_VEL
LIN {X 0,Y 594.259,Z 630.318,A -85,B 0,C 180,E1 -1166.611,E2 -1166.611} C_VEL
LIN {X 0,Y 594.24,Z 633.002,A -85,B 0,C 180,E1 -1167.968,E2 -1167.968} C_VEL
LIN {X 0,Y 594.237,Z 634.333,A -85,B 0,C 180,E1 -1169.323,E2 -1169.323} C_VEL
LIN {X 0,Y 594.237,Z 634.332,A -85,B 0,C 180,E1 -1170.678,E2 -1170.678} C_VEL
LIN {X 0,Y 594.24,Z 632.998,A -85,B 0,C 180,E1 -1172.034,E2 -1172.034} C_VEL
LIN {X 0,Y 594.259,Z 630.313,A -85,B 0,C 180,E1 -1173.391,E2 -1173.391} C_VEL
LIN {X 0,Y 594.237,Z 626.196,A -85,B 0,C 180,E1 -1174.75,E2 -1174.75} C_VEL
LIN {X 0,Y 594.28,Z 620.523,A -85,B 0,C 180,E1 -1176.111,E2 -1176.111} C_VEL
LIN {X 0,Y 594.303,Z 614.121,A -85,B 0,C 180,E1 -1177.304,E2 -1177.304} C_VEL
LIN {X 0,Y 594.324,Z 606.164,A -85,B 0,C 180,E1 -1178.501,E2 -1178.501} C_VEL
LIN {X 0,Y 594.367,Z 597.843,A -85,B 0,C 180,E1 -1179.529,E2 -1179.529} C_VEL
LIN {X 0,Y 594.449,Z 587.828,A -85,B 0,C 180,E1 -1180.56,E2 -1180.56} C_VEL
LIN {X 0,Y 594.525,Z 576.553,A -85,B 0,C 180,E1 -1181.513,E2 -1181.513} C_VEL
LIN {X 0,Y 594.582,Z 564.083,A -85,B 0,C 180,E1 -1182.372,E2 -1182.372} C_VEL
LIN {X 0,Y 594.656,Z 551.621,A -85,B 0,C 180,E1 -1183.064,E2 -1183.064} C_VEL
LIN {X 0,Y 594.743,Z 537.694,A -85,B 0,C 180,E1 -1183.671,E2 -1183.671} C_VEL
LIN {X 0,Y 594.825,Z 523.532,A -85,B 0,C 180,E1 -1184.129,E2 -1184.129} C_VEL
LIN {X 0,Y 594.858,Z 509.846,A -85,B 0,C 180,E1 -1184.432,E2 -1184.432} C_VEL
LIN {X 0,Y 594.916,Z 374.436,A -85,B 0,C 180,E1 -1186.11,E2 -1186.11} C_VEL
LIN {X 0,Y 594.565,Z 372.182,A -85,B 0,C 180,E1 -1186.173,E2 -1186.173} C_VEL
LIN {X 0,Y 594.585,Z 354.006,A -85,B 0,C 180,E1 -1188.612,E2 -1188.612} C_VEL
LIN {X 0,Y 594.715,Z 335.272,A -85,B 0,C 180,E1 -1191.187,E2 -1191.187} C_VEL
LIN {X 0,Y 594.715,Z 326.824,A -85,B 0,C 180,E1 -1192.364,E2 -1192.364} C_VEL
LIN {X 0,Y 594.405,Z 325.163,A -85,B 0,C 180,E1 -1192.659,E2 -1192.659} C_VEL
LIN {X 0,Y 594.378,Z 325.067,A -85,B 0,C 180,E1 -1195.194,E2 -1195.194} C_VEL
LIN {X 0,Y 594.391,Z 325.066,A -85,B 0,C 180,E1 -1197.527,E2 -1197.527} C_VEL
LIN {X 0,Y 594.391,Z 325.072,A -85,B 0,C 180,E1 -1200.329,E2 -1200.329} C_VEL
LIN {X 0,Y 594.381,Z 325.066,A -85,B 0,C 180,E1 -1202.951,E2 -1202.951} C_VEL
LIN {X 0,Y 594.387,Z 325.066,A -85,B 0,C 180,E1 -1205.407,E2 -1205.407} C_VEL
LIN {X 0,Y 594.391,Z 325.074,A -85,B 0,C 180,E1 -1207.941,E2 -1207.941} C_VEL
LIN {X 0,Y 594.378,Z 325.066,A -85,B 0,C 180,E1 -1210.822,E2 -1210.822} C_VEL
LIN {X 0,Y 594.369,Z 325.069,A -85,B 0,C 180,E1 -1213.3,E2 -1213.3} C_VEL
LIN {X 0,Y 594.373,Z 325.072,A -85,B 0,C 180,E1 -1216.161,E2 -1216.161} C_VEL
LIN {X 0,Y 594.384,Z 325.066,A -85,B 0,C 180,E1 -1218.536,E2 -1218.536} C_VEL
LIN {X 0,Y 594.385,Z 325.068,A -85,B 0,C 180,E1 -1221.296,E2 -1221.296} C_VEL
LIN {X 0,Y 594.354,Z 325.079,A -85,B 0,C 180,E1 -1223.756,E2 -1223.756} C_VEL
LIN {X 0,Y 594.38,Z 325.068,A -85,B 0,C 180,E1 -1226.239,E2 -1226.239} C_VEL
LIN {X 0,Y 594.373,Z 325.067,A -85,B 0,C 180,E1 -1228.65,E2 -1228.65} C_VEL
LIN {X 0,Y 594.388,Z 325.068,A -85,B 0,C 180,E1 -1231.042,E2 -1231.042} C_VEL
LIN {X 0,Y 594.386,Z 325.073,A -85,B 0,C 180,E1 -1233.978,E2 -1233.978} C_VEL
LIN {X 0,Y 594.407,Z 325.33,A -85,B 0,C 180,E1 -1235.065,E2 -1235.065} C_VEL
LIN {X 0,Y 594.986,Z 329.093,A -85,B 0,C 180,E1 -1235.58,E2 -1235.58} C_VEL
LIN {X 0,Y 594.842,Z 351.336,A -85,B 0,C 180,E1 -1238.333,E2 -1238.333} C_VEL
LIN {X 0,Y 594.695,Z 375.359,A -85,B 0,C 180,E1 -1241.25,E2 -1241.25} C_VEL
LIN {X 0,Y 594.582,Z 400.273,A -85,B 0,C 180,E1 -1244.225,E2 -1244.225} C_VEL
LIN {X 0,Y 594.476,Z 421.149,A -85,B 0,C 180,E1 -1246.672,E2 -1246.672} C_VEL
LIN {X 0,Y 594.761,Z 424.307,A -85,B 0,C 180,E1 -1246.743,E2 -1246.743} C_VEL
LIN {X 0,Y 594.668,Z 530.329,A -85,B 0,C 180,E1 -1248.042,E2 -1248.042} C_VEL
LIN {X 0,Y 594.632,Z 543.677,A -85,B 0,C 180,E1 -1248.344,E2 -1248.344} C_VEL
LIN {X 0,Y 594.595,Z 555.668,A -85,B 0,C 180,E1 -1248.748,E2 -1248.748} C_VEL
LIN {X 0,Y 594.544,Z 567.257,A -85,B 0,C 180,E1 -1249.27,E2 -1249.27} C_VEL
LIN {X 0,Y 594.471,Z 579.038,A -85,B 0,C 180,E1 -1249.958,E2 -1249.958} C_VEL
LIN {X 0,Y 594.414,Z 589.546,A -85,B 0,C 180,E1 -1250.73,E2 -1250.73} C_VEL
LIN {X 0,Y 594.384,Z 598.152,A -85,B 0,C 180,E1 -1251.501,E2 -1251.501} C_VEL
LIN {X 0,Y 594.347,Z 606.073,A -85,B 0,C 180,E1 -1252.355,E2 -1252.355} C_VEL
LIN {X 0,Y 594.306,Z 613.898,A -85,B 0,C 180,E1 -1253.39,E2 -1253.39} C_VEL
LIN {X 0,Y 594.289,Z 620.944,A -85,B 0,C 180,E1 -1254.571,E2 -1254.571} C_VEL
LIN {X 0,Y 594.27,Z 625.686,A -85,B 0,C 180,E1 -1255.591,E2 -1255.591} C_VEL
LIN {X 0,Y 594.268,Z 629.317,A -85,B 0,C 180,E1 -1256.61,E2 -1256.61} C_VEL
LIN {X 0,Y 594.225,Z 631.192,A -85,B 0,C 180,E1 -1257.288,E2 -1257.288} C_VEL
LIN {X 0,Y 594.24,Z 632.627,A -85,B 0,C 180,E1 -1257.967,E2 -1257.967} C_VEL
LIN {X 0,Y 594.24,Z 634.253,A -85,B 0,C 180,E1 -1259.322,E2 -1259.322} C_VEL
LIN {X 0,Y 594.236,Z 634.496,A -85,B 0,C 180,E1 -1260,E2 -1260} C_VEL
LIN {X 0,Y 594.24,Z 634.315,A -85,B 0,C 180,E1 -1260.678,E2 -1260.678} C_VEL
LIN {X 0,Y 594.239,Z 632.773,A -85,B 0,C 180,E1 -1262.033,E2 -1262.033} C_VEL
LIN {X 0,Y 594.226,Z 631.415,A -85,B 0,C 180,E1 -1262.712,E2 -1262.712} C_VEL
LIN {X 0,Y 594.289,Z 628.54,A -85,B 0,C 180,E1 -1263.729,E2 -1263.729} C_VEL
LIN {X 0,Y 594.242,Z 624.641,A -85,B 0,C 180,E1 -1264.749,E2 -1264.749} C_VEL
LIN {X 0,Y 594.299,Z 619.61,A -85,B 0,C 180,E1 -1265.769,E2 -1265.769} C_VEL
LIN {X 0,Y 594.317,Z 613.283,A -85,B 0,C 180,E1 -1266.791,E2 -1266.791} C_VEL
LIN {X 0,Y 594.347,Z 605.375,A -85,B 0,C 180,E1 -1267.816,E2 -1267.816} C_VEL
LIN {X 0,Y 594.381,Z 595.521,A -85,B 0,C 180,E1 -1268.842,E2 -1268.842} C_VEL
LIN {X 0,Y 594.423,Z 585.205,A -85,B 0,C 180,E1 -1269.7,E2 -1269.7} C_VEL
LIN {X 0,Y 594.504,Z 573.59,A -85,B 0,C 180,E1 -1270.472,E2 -1270.472} C_VEL
LIN {X 0,Y 594.571,Z 561.678,A -85,B 0,C 180,E1 -1271.089,E2 -1271.089} C_VEL
LIN {X 0,Y 594.619,Z 548.744,A -85,B 0,C 180,E1 -1271.591,E2 -1271.591} C_VEL
LIN {X 0,Y 594.652,Z 541.22,A -85,B 0,C 180,E1 -1271.814,E2 -1271.814} C_VEL
LIN {X 0,Y 593.923,Z 535.552,A -85,B 0,C 180,E1 -1271.963,E2 -1271.963} C_VEL
LIN {X 0,Y 588.802,Z 518.868,A -85,B 0,C 180,E1 -1272.328,E2 -1272.328} C_VEL
LIN {X 0,Y 587.838,Z 513.115,A -85,B 0,C 180,E1 -1272.416,E2 -1272.416} C_VEL
LIN {X 0,Y 587.772,Z 511.164,A -85,B 0,C 180,E1 -1272.441,E2 -1272.441} C_VEL
LIN {X 0,Y 587.783,Z 423.608,A -85,B 0,C 180,E1 -1273.516,E2 -1273.516} C_VEL
LIN {X 0,Y 587.459,Z 421.179,A -85,B 0,C 180,E1 -1273.579,E2 -1273.579} C_VEL
LIN {X 0,Y 587.587,Z 398.059,A -85,B 0,C 180,E1 -1276.325,E2 -1276.325} C_VEL
LIN {X 0,Y 587.754,Z 375.689,A -85,B 0,C 180,E1 -1279.03,E2 -1279.03} C_VEL
LIN {X 0,Y 587.977,Z 352.063,A -85,B 0,C 180,E1 -1281.933,E2 -1281.933} C_VEL
LIN {X 0,Y 588.14,Z 330.793,A -85,B 0,C 180,E1 -1284.598,E2 -1284.598} C_VEL
LIN {X 0,Y 587.376,Z 326.245,A -85,B 0,C 180,E1 -1285.23,E2 -1285.23} C_VEL
LIN {X 0,Y 587.332,Z 325.952,A -85,B 0,C 180,E1 -1285.517,E2 -1285.517} C_VEL
LIN {X 0,Y 587.345,Z 325.945,A -85,B 0,C 180,E1 -1287.818,E2 -1287.818} C_VEL
LIN {X 0,Y 587.34,Z 325.953,A -85,B 0,C 180,E1 -1290.509,E2 -1290.509} C_VEL
LIN {X 0,Y 587.338,Z 325.943,A -85,B 0,C 180,E1 -1293.397,E2 -1293.397} C_VEL
LIN {X 0,Y 587.294,Z 325.952,A -85,B 0,C 180,E1 -1295.9,E2 -1295.9} C_VEL
LIN {X 0,Y 587.331,Z 325.951,A -85,B 0,C 180,E1 -1298.479,E2 -1298.479} C_VEL
LIN {X 0,Y 587.339,Z 325.943,A -85,B 0,C 180,E1 -1301.157,E2 -1301.157} C_VEL
LIN {X 0,Y 587.333,Z 325.952,A -85,B 0,C 180,E1 -1304.113,E2 -1304.113} C_VEL
LIN {X 0,Y 587.316,Z 325.946,A -85,B 0,C 180,E1 -1306.993,E2 -1306.993} C_VEL
LIN {X 0,Y 587.316,Z 325.95,A -85,B 0,C 180,E1 -1309.745,E2 -1309.745} C_VEL
LIN {X 0,Y 587.349,Z 325.946,A -85,B 0,C 180,E1 -1312.392,E2 -1312.392} C_VEL
LIN {X 0,Y 587.361,Z 325.945,A -85,B 0,C 180,E1 -1315.651,E2 -1315.651} C_VEL
LIN {X 0,Y 587.345,Z 325.948,A -85,B 0,C 180,E1 -1318.231,E2 -1318.231} C_VEL
LIN {X 0,Y 587.355,Z 325.938,A -85,B 0,C 180,E1 -1320.866,E2 -1320.866} C_VEL
LIN {X 0,Y 587.364,Z 325.947,A -85,B 0,C 180,E1 -1323.819,E2 -1323.819} C_VEL
LIN {X 0,Y 587.342,Z 325.95,A -85,B 0,C 180,E1 -1325.993,E2 -1325.993} C_VEL
LIN {X 0,Y 587.351,Z 326.119,A -85,B 0,C 180,E1 -1327.258,E2 -1327.258} C_VEL
LIN {X 0,Y 587.858,Z 330.15,A -85,B 0,C 180,E1 -1327.877,E2 -1327.877} C_VEL
LIN {X 0,Y 587.691,Z 350.447,A -85,B 0,C 180,E1 -1330.713,E2 -1330.713} C_VEL
LIN {X 0,Y 587.542,Z 370.676,A -85,B 0,C 180,E1 -1333.495,E2 -1333.495} C_VEL
LIN {X 0,Y 587.586,Z 372.186,A -85,B 0,C 180,E1 -1333.675,E2 -1333.675} C_VEL
LIN {X 0,Y 588.196,Z 377.308,A -85,B 0,C 180,E1 -1333.781,E2 -1333.781} C_VEL
LIN {X 0,Y 588.001,Z 508.329,A -85,B 0,C 180,E1 -1335.418,E2 -1335.418} C_VEL
LIN {X 0,Y 587.929,Z 521.621,A -85,B 0,C 180,E1 -1335.698,E2 -1335.698} C_VEL
LIN {X 0,Y 587.84,Z 536.547,A -85,B 0,C 180,E1 -1336.165,E2 -1336.165} C_VEL
LIN {X 0,Y 587.756,Z 548.922,A -85,B 0,C 180,E1 -1336.692,E2 -1336.692} C_VEL
LIN {X 0,Y 587.657,Z 560.455,A -85,B 0,C 180,E1 -1337.305,E2 -1337.305} C_VEL
LIN {X 0,Y 587.574,Z 571.27,A -85,B 0,C 180,E1 -1338.004,E2 -1338.004} C_VEL
LIN {X 0,Y 587.472,Z 581.626,A -85,B 0,C 180,E1 -1338.807,E2 -1338.807} C_VEL
LIN {X 0,Y 587.377,Z 592.661,A -85,B 0,C 180,E1 -1339.834,E2 -1339.834} C_VEL
LIN {X 0,Y 587.339,Z 601.832,A -85,B 0,C 180,E1 -1340.877,E2 -1340.877} C_VEL
LIN {X 0,Y 587.27,Z 609.477,A -85,B 0,C 180,E1 -1341.916,E2 -1341.916} C_VEL
LIN {X 0,Y 587.211,Z 616.805,A -85,B 0,C 180,E1 -1343.125,E2 -1343.125} C_VEL
LIN {X 0,Y 587.227,Z 621.902,A -85,B 0,C 180,E1 -1344.16,E2 -1344.16} C_VEL
LIN {X 0,Y 587.186,Z 627.246,A -85,B 0,C 180,E1 -1345.537,E2 -1345.537} C_VEL
LIN {X 0,Y 587.182,Z 630.201,A -85,B 0,C 180,E1 -1346.568,E2 -1346.568} C_VEL
LIN {X 0,Y 587.14,Z 632.935,A -85,B 0,C 180,E1 -1347.941,E2 -1347.941} C_VEL
LIN {X 0,Y 587.135,Z 634.296,A -85,B 0,C 180,E1 -1349.313,E2 -1349.313} C_VEL
LIN {X 0,Y 587.137,Z 634.332,A -85,B 0,C 180,E1 -1350.685,E2 -1350.685} C_VEL
LIN {X 0,Y 587.139,Z 633.075,A -85,B 0,C 180,E1 -1352.057,E2 -1352.057} C_VEL
LIN {X 0,Y 587.182,Z 630.437,A -85,B 0,C 180,E1 -1353.43,E2 -1353.43} C_VEL
LIN {X 0,Y 587.14,Z 626.352,A -85,B 0,C 180,E1 -1354.805,E2 -1354.805} C_VEL
LIN {X 0,Y 587.227,Z 622.319,A -85,B 0,C 180,E1 -1355.838,E2 -1355.838} C_VEL
LIN {X 0,Y 587.209,Z 617.296,A -85,B 0,C 180,E1 -1356.873,E2 -1356.873} C_VEL
LIN {X 0,Y 587.269,Z 610.076,A -85,B 0,C 180,E1 -1358.083,E2 -1358.083} C_VEL
LIN {X 0,Y 587.316,Z 601.191,A -85,B 0,C 180,E1 -1359.296,E2 -1359.296} C_VEL
LIN {X 0,Y 587.371,Z 591.849,A -85,B 0,C 180,E1 -1360.338,E2 -1360.338} C_VEL
LIN {X 0,Y 587.478,Z 581.471,A -85,B 0,C 180,E1 -1361.296,E2 -1361.296} C_VEL
LIN {X 0,Y 587.57,Z 570.091,A -85,B 0,C 180,E1 -1362.169,E2 -1362.169} C_VEL
LIN {X 0,Y 587.668,Z 557.483,A -85,B 0,C 180,E1 -1362.957,E2 -1362.957} C_VEL
LIN {X 0,Y 587.801,Z 543.205,A -85,B 0,C 180,E1 -1363.658,E2 -1363.658} C_VEL
LIN {X 0,Y 587.922,Z 530.06,A -85,B 0,C 180,E1 -1364.146,E2 -1364.146} C_VEL
LIN {X 0,Y 587.954,Z 516.816,A -85,B 0,C 180,E1 -1364.508,E2 -1364.508} C_VEL
LIN {X 0,Y 588.037,Z 502.731,A -85,B 0,C 180,E1 -1364.756,E2 -1364.756} C_VEL
LIN {X 0,Y 588.156,Z 375.729,A -85,B 0,C 180,E1 -1366.33,E2 -1366.33} C_VEL
LIN {X 0,Y 587.572,Z 372.216,A -85,B 0,C 180,E1 -1366.413,E2 -1366.413} C_VEL
LIN {X 0,Y 587.679,Z 352.2,A -85,B 0,C 180,E1 -1369.134,E2 -1369.134} C_VEL
LIN {X 0,Y 587.874,Z 330.8,A -85,B 0,C 180,E1 -1372.121,E2 -1372.121} C_VEL
LIN {X 0,Y 587.401,Z 326.306,A -85,B 0,C 180,E1 -1372.791,E2 -1372.791} C_VEL
LIN {X 0,Y 587.333,Z 326.041,A -85,B 0,C 180,E1 -1372.871,E2 -1372.871} C_VEL
LIN {X 0,Y 587.336,Z 325.945,A -85,B 0,C 180,E1 -1375.515,E2 -1375.515} C_VEL
LIN {X 0,Y 587.348,Z 325.947,A -85,B 0,C 180,E1 -1377.816,E2 -1377.816} C_VEL
LIN {X 0,Y 587.35,Z 325.946,A -85,B 0,C 180,E1 -1380.512,E2 -1380.512} C_VEL
LIN {X 0,Y 587.333,Z 325.944,A -85,B 0,C 180,E1 -1383.395,E2 -1383.395} C_VEL
LIN {X 0,Y 587.354,Z 325.948,A -85,B 0,C 180,E1 -1385.894,E2 -1385.894} C_VEL
LIN {X 0,Y 587.331,Z 325.946,A -85,B 0,C 180,E1 -1388.478,E2 -1388.478} C_VEL
LIN {X 0,Y 587.335,Z 325.943,A -85,B 0,C 180,E1 -1391.155,E2 -1391.155} C_VEL
LIN {X 0,Y 587.328,Z 325.949,A -85,B 0,C 180,E1 -1394.113,E2 -1394.113} C_VEL
LIN {X 0,Y 587.33,Z 325.943,A -85,B 0,C 180,E1 -1396.995,E2 -1396.995} C_VEL
LIN {X 0,Y 587.322,Z 325.955,A -85,B 0,C 180,E1 -1399.746,E2 -1399.746} C_VEL
LIN {X 0,Y 587.34,Z 325.941,A -85,B 0,C 180,E1 -1402.392,E2 -1402.392} C_VEL
LIN {X 0,Y 587.34,Z 325.943,A -85,B 0,C 180,E1 -1404.945,E2 -1404.945} C_VEL
LIN {X 0,Y 587.336,Z 325.95,A -85,B 0,C 180,E1 -1407.421,E2 -1407.421} C_VEL
LIN {X 0,Y 587.338,Z 325.945,A -85,B 0,C 180,E1 -1409.83,E2 -1409.83} C_VEL
LIN {X 0,Y 587.343,Z 325.941,A -85,B 0,C 180,E1 -1412.306,E2 -1412.306} C_VEL
LIN {X 0,Y 587.33,Z 325.943,A -85,B 0,C 180,E1 -1414.483,E2 -1414.483} C_VEL
LIN {X 0,Y 587.361,Z 325.949,A -85,B 0,C 180,E1 -1417.487,E2 -1417.487} C_VEL
LIN {X 0,Y 587.339,Z 325.942,A -85,B 0,C 180,E1 -1420.425,E2 -1420.425} C_VEL
LIN {X 0,Y 587.351,Z 325.951,A -85,B 0,C 180,E1 -1423.311,E2 -1423.311} C_VEL
LIN {X 0,Y 587.352,Z 325.941,A -85,B 0,C 180,E1 -1426.154,E2 -1426.154} C_VEL
LIN {X 0,Y 587.343,Z 325.948,A -85,B 0,C 180,E1 -1428.962,E2 -1428.962} C_VEL
LIN {X 0,Y 587.364,Z 325.941,A -85,B 0,C 180,E1 -1431.745,E2 -1431.745} C_VEL
LIN {X 0,Y 587.357,Z 325.942,A -85,B 0,C 180,E1 -1434.507,E2 -1434.507} C_VEL
LIN {X 0,Y 587.378,Z 325.944,A -85,B 0,C 180,E1 -1437.257,E2 -1437.257} C_VEL
LIN {X 0,Y 587.373,Z 325.938,A -85,B 0,C 180,E1 -1440,E2 -1440} C_VEL
LIN {X 0,Y 587.378,Z 325.944,A -85,B 0,C 180,E1 -1442.743,E2 -1442.743} C_VEL
LIN {X 0,Y 587.357,Z 325.942,A -85,B 0,C 180,E1 -1445.493,E2 -1445.493} C_VEL
LIN {X 0,Y 587.364,Z 325.941,A -85,B 0,C 180,E1 -1448.255,E2 -1448.255} C_VEL
LIN {X 0,Y 587.351,Z 325.946,A -85,B 0,C 180,E1 -1451.142,E2 -1451.142} C_VEL
LIN {X 0,Y 587.355,Z 325.943,A -85,B 0,C 180,E1 -1454.261,E2 -1454.261} C_VEL
LIN {X 0,Y 587.353,Z 325.941,A -85,B 0,C 180,E1 -1457.406,E2 -1457.406} C_VEL
LIN {X 0,Y 587.329,Z 325.948,A -85,B 0,C 180,E1 -1460.305,E2 -1460.305} C_VEL
LIN {X 0,Y 587.358,Z 325.941,A -85,B 0,C 180,E1 -1463.257,E2 -1463.257} C_VEL
LIN {X 0,Y 587.354,Z 325.946,A -85,B 0,C 180,E1 -1466.278,E2 -1466.278} C_VEL
LIN {X 0,Y 587.345,Z 325.939,A -85,B 0,C 180,E1 -1469.135,E2 -1469.135} C_VEL
LIN {X 0,Y 587.351,Z 325.942,A -85,B 0,C 180,E1 -1471.839,E2 -1471.839} C_VEL
LIN {X 0,Y 587.347,Z 325.952,A -85,B 0,C 180,E1 -1474.35,E2 -1474.35} C_VEL
LIN {X 0,Y 587.345,Z 325.943,A -85,B 0,C 180,E1 -1476.747,E2 -1476.747} C_VEL
LIN {X 0,Y 587.339,Z 325.942,A -85,B 0,C 180,E1 -1479.36,E2 -1479.36} C_VEL
LIN {X 0,Y 587.359,Z 325.949,A -85,B 0,C 180,E1 -1482.112,E2 -1482.112} C_VEL
LIN {X 0,Y 587.308,Z 325.945,A -85,B 0,C 180,E1 -1485.09,E2 -1485.09} C_VEL
LIN {X 0,Y 587.346,Z 325.949,A -85,B 0,C 180,E1 -1487.929,E2 -1487.929} C_VEL
LIN {X 0,Y 587.331,Z 325.943,A -85,B 0,C 180,E1 -1491.059,E2 -1491.059} C_VEL
LIN {X 0,Y 587.35,Z 325.942,A -85,B 0,C 180,E1 -1493.292,E2 -1493.292} C_VEL
LIN {X 0,Y 587.367,Z 325.947,A -85,B 0,C 180,E1 -1495.782,E2 -1495.782} C_VEL
LIN {X 0,Y 587.351,Z 325.947,A -85,B 0,C 180,E1 -1498.233,E2 -1498.233} C_VEL
LIN {X 0,Y 587.35,Z 325.938,A -85,B 0,C 180,E1 -1500.867,E2 -1500.867} C_VEL
LIN {X 0,Y 587.359,Z 325.947,A -85,B 0,C 180,E1 -1503.819,E2 -1503.819} C_VEL
LIN {X 0,Y 587.338,Z 325.951,A -85,B 0,C 180,E1 -1505.995,E2 -1505.995} C_VEL
LIN {X 0,Y 587.356,Z 326.163,A -85,B 0,C 180,E1 -1507.225,E2 -1507.225} C_VEL
LIN {X 0,Y 587.867,Z 330.482,A -85,B 0,C 180,E1 -1507.879,E2 -1507.879} C_VEL
LIN {X 0,Y 587.68,Z 351.872,A -85,B 0,C 180,E1 -1510.866,E2 -1510.866} C_VEL
LIN {X 0,Y 587.554,Z 371.721,A -85,B 0,C 180,E1 -1513.586,E2 -1513.586} C_VEL
LIN {X 0,Y 587.716,Z 373.205,A -85,B 0,C 180,E1 -1513.669,E2 -1513.669} C_VEL
LIN {X 0,Y 588.177,Z 377.488,A -85,B 0,C 180,E1 -1513.738,E2 -1513.738} C_VEL
LIN {X 0,Y 587.986,Z 509.937,A -85,B 0,C 180,E1 -1515.398,E2 -1515.398} C_VEL
LIN {X 0,Y 587.934,Z 524.152,A -85,B 0,C 180,E1 -1515.72,E2 -1515.72} C_VEL
LIN {X 0,Y 587.817,Z 537.735,A -85,B 0,C 180,E1 -1516.166,E2 -1516.166} C_VEL
LIN {X 0,Y 587.731,Z 551.66,A -85,B 0,C 180,E1 -1516.781,E2 -1516.781} C_VEL
LIN {X 0,Y 587.626,Z 564.114,A -85,B 0,C 180,E1 -1517.481,E2 -1517.481} C_VEL
LIN {X 0,Y 587.512,Z 576.651,A -85,B 0,C 180,E1 -1518.355,E2 -1518.355} C_VEL
LIN {X 0,Y 587.444,Z 587.846,A -85,B 0,C 180,E1 -1519.314,E2 -1519.314} C_VEL
LIN {X 0,Y 587.319,Z 597.859,A -85,B 0,C 180,E1 -1520.357,E2 -1520.357} C_VEL
LIN {X 0,Y 587.277,Z 606.178,A -85,B 0,C 180,E1 -1521.398,E2 -1521.398} C_VEL
LIN {X 0,Y 587.243,Z 614.132,A -85,B 0,C 180,E1 -1522.609,E2 -1522.609} C_VEL
LIN {X 0,Y 587.202,Z 620.531,A -85,B 0,C 180,E1 -1523.817,E2 -1523.817} C_VEL
LIN {X 0,Y 587.16,Z 624.964,A -85,B 0,C 180,E1 -1524.85,E2 -1524.85} C_VEL
LIN {X 0,Y 587.179,Z 628.446,A -85,B 0,C 180,E1 -1525.883,E2 -1525.883} C_VEL
LIN {X 0,Y 587.13,Z 631.834,A -85,B 0,C 180,E1 -1527.257,E2 -1527.257} C_VEL
LIN {X 0,Y 587.141,Z 633.833,A -85,B 0,C 180,E1 -1528.629,E2 -1528.629} C_VEL
LIN {X 0,Y 587.135,Z 634.5,A -85,B 0,C 180,E1 -1530.001,E2 -1530.001} C_VEL
LIN {X 0,Y 587.141,Z 633.831,A -85,B 0,C 180,E1 -1531.373,E2 -1531.373} C_VEL
LIN {X 0,Y 587.13,Z 631.83,A -85,B 0,C 180,E1 -1532.745,E2 -1532.745} C_VEL
LIN {X 0,Y 587.179,Z 628.44,A -85,B 0,C 180,E1 -1534.119,E2 -1534.119} C_VEL
LIN {X 0,Y 587.199,Z 623.565,A -85,B 0,C 180,E1 -1535.495,E2 -1535.495} C_VEL
LIN {X 0,Y 587.21,Z 617.048,A -85,B 0,C 180,E1 -1536.875,E2 -1536.875} C_VEL
LIN {X 0,Y 587.269,Z 609.794,A -85,B 0,C 180,E1 -1538.084,E2 -1538.084} C_VEL
LIN {X 0,Y 587.322,Z 600.816,A -85,B 0,C 180,E1 -1539.297,E2 -1539.297} C_VEL
LIN {X 0,Y 587.372,Z 591.383,A -85,B 0,C 180,E1 -1540.34,E2 -1540.34} C_VEL
LIN {X 0,Y 587.476,Z 581.021,A -85,B 0,C 180,E1 -1541.291,E2 -1541.291} C_VEL
LIN {X 0,Y 587.575,Z 569.419,A -85,B 0,C 180,E1 -1542.171,E2 -1542.171} C_VEL
LIN {X 0,Y 587.672,Z 556.633,A -85,B 0,C 180,E1 -1542.958,E2 -1542.958} C_VEL
LIN {X 0,Y 587.8,Z 544.143,A -85,B 0,C 180,E1 -1543.571,E2 -1543.571} C_VEL
LIN {X 0,Y 587.919,Z 530.588,A -85,B 0,C 180,E1 -1544.086,E2 -1544.086} C_VEL
LIN {X 0,Y 587.949,Z 516.923,A -85,B 0,C 180,E1 -1544.462,E2 -1544.462} C_VEL
LIN {X 0,Y 588.02,Z 502.544,A -85,B 0,C 180,E1 -1544.714,E2 -1544.714} C_VEL
LIN {X 0,Y 588.123,Z 375.553,A -85,B 0,C 180,E1 -1546.288,E2 -1546.288} C_VEL
LIN {X 0,Y 587.562,Z 372.19,A -85,B 0,C 180,E1 -1546.371,E2 -1546.371} C_VEL
LIN {X 0,Y 587.651,Z 352.762,A -85,B 0,C 180,E1 -1549.012,E2 -1549.012} C_VEL
LIN {X 0,Y 587.854,Z 333.084,A -85,B 0,C 180,E1 -1551.754,E2 -1551.754} C_VEL
LIN {X 0,Y 587.73,Z 327.853,A -85,B 0,C 180,E1 -1552.499,E2 -1552.499} C_VEL
LIN {X 0,Y 587.359,Z 326.099,A -85,B 0,C 180,E1 -1552.792,E2 -1552.792} C_VEL
LIN {X 0,Y 587.338,Z 325.945,A -85,B 0,C 180,E1 -1555.517,E2 -1555.517} C_VEL
LIN {X 0,Y 587.354,Z 325.947,A -85,B 0,C 180,E1 -1557.818,E2 -1557.818} C_VEL
LIN {X 0,Y 587.342,Z 325.947,A -85,B 0,C 180,E1 -1560.51,E2 -1560.51} C_VEL
LIN {X 0,Y 587.338,Z 325.944,A -85,B 0,C 180,E1 -1563.397,E2 -1563.397} C_VEL
LIN {X 0,Y 587.361,Z 325.949,A -85,B 0,C 180,E1 -1565.896,E2 -1565.896} C_VEL
LIN {X 0,Y 587.334,Z 325.947,A -85,B 0,C 180,E1 -1568.48,E2 -1568.48} C_VEL
LIN {X 0,Y 587.339,Z 325.943,A -85,B 0,C 180,E1 -1571.157,E2 -1571.157} C_VEL
LIN {X 0,Y 587.316,Z 325.952,A -85,B 0,C 180,E1 -1574.112,E2 -1574.112} C_VEL
LIN {X 0,Y 587.319,Z 325.946,A -85,B 0,C 180,E1 -1576.994,E2 -1576.994} C_VEL
LIN {X 0,Y 587.315,Z 325.956,A -85,B 0,C 180,E1 -1579.746,E2 -1579.746} C_VEL
LIN {X 0,Y 587.348,Z 325.943,A -85,B 0,C 180,E1 -1582.393,E2 -1582.393} C_VEL
LIN {X 0,Y 587.362,Z 325.949,A -85,B 0,C 180,E1 -1585.78,E2 -1585.78} C_VEL
LIN {X 0,Y 587.346,Z 325.944,A -85,B 0,C 180,E1 -1588.231,E2 -1588.231} C_VEL
LIN {X 0,Y 587.354,Z 325.943,A -85,B 0,C 180,E1 -1590.867,E2 -1590.867} C_VEL
LIN {X 0,Y 587.362,Z 325.949,A -85,B 0,C 180,E1 -1593.82,E2 -1593.82} C_VEL
LIN {X 0,Y 587.378,Z 326.16,A -85,B 0,C 180,E1 -1594.841,E2 -1594.841} C_VEL
LIN {X 0,Y 588.135,Z 330.257,A -85,B 0,C 180,E1 -1595.424,E2 -1595.424} C_VEL
LIN {X 0,Y 587.974,Z 351.34,A -85,B 0,C 180,E1 -1598.067,E2 -1598.067} C_VEL
LIN {X 0,Y 587.783,Z 374.879,A -85,B 0,C 180,E1 -1600.962,E2 -1600.962} C_VEL
LIN {X 0,Y 587.619,Z 400.278,A -85,B 0,C 180,E1 -1604.033,E2 -1604.033} C_VEL
LIN {X 0,Y 587.498,Z 421.156,A -85,B 0,C 180,E1 -1606.51,E2 -1606.51} C_VEL
LIN {X 0,Y 587.856,Z 426.141,A -85,B 0,C 180,E1 -1606.607,E2 -1606.607} C_VEL
LIN {X 0,Y 587.723,Z 530.347,A -85,B 0,C 180,E1 -1607.899,E2 -1607.899} C_VEL
LIN {X 0,Y 587.702,Z 543.705,A -85,B 0,C 180,E1 -1608.205,E2 -1608.205} C_VEL
LIN {X 0,Y 587.63,Z 556.259,A -85,B 0,C 180,E1 -1608.635,E2 -1608.635} C_VEL
LIN {X 0,Y 587.537,Z 568.916,A -85,B 0,C 180,E1 -1609.228,E2 -1609.228} C_VEL
LIN {X 0,Y 587.455,Z 580.327,A -85,B 0,C 180,E1 -1609.923,E2 -1609.923} C_VEL
LIN {X 0,Y 587.384,Z 590.602,A -85,B 0,C 180,E1 -1610.705,E2 -1610.705} C_VEL
LIN {X 0,Y 587.341,Z 599.875,A -85,B 0,C 180,E1 -1611.571,E2 -1611.571} C_VEL
LIN {X 0,Y 587.26,Z 608.844,A -85,B 0,C 180,E1 -1612.608,E2 -1612.608} C_VEL
LIN {X 0,Y 587.199,Z 615.939,A -85,B 0,C 180,E1 -1613.625,E2 -1613.625} C_VEL
LIN {X 0,Y 587.211,Z 620.949,A -85,B 0,C 180,E1 -1614.506,E2 -1614.506} C_VEL
LIN {X 0,Y 587.188,Z 625.69,A -85,B 0,C 180,E1 -1615.538,E2 -1615.538} C_VEL
LIN {X 0,Y 587.195,Z 629.32,A -85,B 0,C 180,E1 -1616.569,E2 -1616.569} C_VEL
LIN {X 0,Y 587.132,Z 631.193,A -85,B 0,C 180,E1 -1617.256,E2 -1617.256} C_VEL
LIN {X 0,Y 587.139,Z 632.628,A -85,B 0,C 180,E1 -1617.942,E2 -1617.942} C_VEL
LIN {X 0,Y 587.14,Z 634.253,A -85,B 0,C 180,E1 -1619.314,E2 -1619.314} C_VEL
LIN {X 0,Y 587.137,Z 634.496,A -85,B 0,C 180,E1 -1620,E2 -1620} C_VEL
LIN {X 0,Y 587.14,Z 634.314,A -85,B 0,C 180,E1 -1620.686,E2 -1620.686} C_VEL
LIN {X 0,Y 587.138,Z 632.772,A -85,B 0,C 180,E1 -1622.058,E2 -1622.058} C_VEL
LIN {X 0,Y 587.133,Z 631.414,A -85,B 0,C 180,E1 -1622.744,E2 -1622.744} C_VEL
LIN {X 0,Y 587.213,Z 628.539,A -85,B 0,C 180,E1 -1623.774,E2 -1623.774} C_VEL
LIN {X 0,Y 587.147,Z 624.64,A -85,B 0,C 180,E1 -1624.806,E2 -1624.806} C_VEL
LIN {X 0,Y 587.229,Z 619.61,A -85,B 0,C 180,E1 -1625.839,E2 -1625.839} C_VEL
LIN {X 0,Y 587.23,Z 613.277,A -85,B 0,C 180,E1 -1626.874,E2 -1626.874} C_VEL
LIN {X 0,Y 587.288,Z 605.372,A -85,B 0,C 180,E1 -1627.91,E2 -1627.91} C_VEL
LIN {X 0,Y 587.336,Z 597.303,A -85,B 0,C 180,E1 -1628.776,E2 -1628.776} C_VEL
LIN {X 0,Y 587.386,Z 587.467,A -85,B 0,C 180,E1 -1629.643,E2 -1629.643} C_VEL
LIN {X 0,Y 587.484,Z 576.41,A -85,B 0,C 180,E1 -1630.425,E2 -1630.425} C_VEL
LIN {X 0,Y 587.578,Z 564.004,A -85,B 0,C 180,E1 -1631.112,E2 -1631.112} C_VEL
LIN {X 0,Y 587.643,Z 551.387,A -85,B 0,C 180,E1 -1631.64,E2 -1631.64} C_VEL
LIN {X 0,Y 587.717,Z 537.938,A -85,B 0,C 180,E1 -1632.036,E2 -1632.036} C_VEL
LIN {X 0,Y 587.76,Z 524.664,A -85,B 0,C 180,E1 -1632.276,E2 -1632.276} C_VEL
LIN {X 0,Y 587.772,Z 511.164,A -85,B 0,C 180,E1 -1632.441,E2 -1632.441} C_VEL
LIN {X 0,Y 587.155,Z 505.355,A -85,B 0,C 180,E1 -1632.526,E2 -1632.526} C_VEL
LIN {X 0,Y 581.567,Z 486.659,A -85,B 0,C 180,E1 -1632.879,E2 -1632.879} C_VEL
LIN {X 0,Y 580.904,Z 480.85,A -85,B 0,C 180,E1 -1632.966,E2 -1632.966} C_VEL
LIN {X 0,Y 580.815,Z 423.785,A -85,B 0,C 180,E1 -1633.679,E2 -1633.679} C_VEL
LIN {X 0,Y 580.48,Z 421.171,A -85,B 0,C 180,E1 -1633.745,E2 -1633.745} C_VEL
LIN {X 0,Y 580.64,Z 398.054,A -85,B 0,C 180,E1 -1636.526,E2 -1636.526} C_VEL
LIN {X 0,Y 580.819,Z 375.438,A -85,B 0,C 180,E1 -1639.297,E2 -1639.297} C_VEL
LIN {X 0,Y 581.087,Z 353.542,A -85,B 0,C 180,E1 -1642.02,E2 -1642.02} C_VEL
LIN {X 0,Y 581.303,Z 333.226,A -85,B 0,C 180,E1 -1644.589,E2 -1644.589} C_VEL
LIN {X 0,Y 580.534,Z 328.046,A -85,B 0,C 180,E1 -1645.261,E2 -1645.261} C_VEL
LIN {X 0,Y 580.294,Z 326.913,A -85,B 0,C 180,E1 -1645.464,E2 -1645.464} C_VEL
LIN {X 0,Y 580.302,Z 326.826,A -85,B 0,C 180,E1 -1648.186,E2 -1648.186} C_VEL
LIN {X 0,Y 580.288,Z 326.828,A -85,B 0,C 180,E1 -1650.694,E2 -1650.694} C_VEL
LIN {X 0,Y 580.308,Z 326.819,A -85,B 0,C 180,E1 -1653.316,E2 -1653.316} C_VEL
LIN {X 0,Y 580.249,Z 326.828,A -85,B 0,C 180,E1 -1655.756,E2 -1655.756} C_VEL
LIN {X 0,Y 580.292,Z 326.828,A -85,B 0,C 180,E1 -1658.146,E2 -1658.146} C_VEL
LIN {X 0,Y 580.301,Z 326.822,A -85,B 0,C 180,E1 -1660.843,E2 -1660.843} C_VEL
LIN {X 0,Y 580.285,Z 326.823,A -85,B 0,C 180,E1 -1663.658,E2 -1663.658} C_VEL
LIN {X 0,Y 580.278,Z 326.826,A -85,B 0,C 180,E1 -1666.61,E2 -1666.61} C_VEL
LIN {X 0,Y 580.301,Z 326.819,A -85,B 0,C 180,E1 -1669.156,E2 -1669.156} C_VEL
LIN {X 0,Y 580.295,Z 326.828,A -85,B 0,C 180,E1 -1671.927,E2 -1671.927} C_VEL
LIN {X 0,Y 580.29,Z 326.824,A -85,B 0,C 180,E1 -1674.455,E2 -1674.455} C_VEL
LIN {X 0,Y 580.294,Z 326.82,A -85,B 0,C 180,E1 -1676.975,E2 -1676.975} C_VEL
LIN {X 0,Y 580.302,Z 326.823,A -85,B 0,C 180,E1 -1679.425,E2 -1679.425} C_VEL
LIN {X 0,Y 580.303,Z 326.826,A -85,B 0,C 180,E1 -1682.141,E2 -1682.141} C_VEL
LIN {X 0,Y 580.327,Z 326.82,A -85,B 0,C 180,E1 -1685.269,E2 -1685.269} C_VEL
LIN {X 0,Y 580.324,Z 327.042,A -85,B 0,C 180,E1 -1687.105,E2 -1687.105} C_VEL
LIN {X 0,Y 580.955,Z 331.462,A -85,B 0,C 180,E1 -1687.787,E2 -1687.787} C_VEL
LIN {X 0,Y 580.741,Z 352.237,A -85,B 0,C 180,E1 -1690.724,E2 -1690.724} C_VEL
LIN {X 0,Y 580.566,Z 371.72,A -85,B 0,C 180,E1 -1693.426,E2 -1693.426} C_VEL
LIN {X 0,Y 580.687,Z 373.03,A -85,B 0,C 180,E1 -1693.506,E2 -1693.506} C_VEL
LIN {X 0,Y 581.404,Z 377.354,A -85,B 0,C 180,E1 -1693.586,E2 -1693.586} C_VEL
LIN {X 0,Y 581.141,Z 508.307,A -85,B 0,C 180,E1 -1695.242,E2 -1695.242} C_VEL
LIN {X 0,Y 581.031,Z 521.351,A -85,B 0,C 180,E1 -1695.518,E2 -1695.518} C_VEL
LIN {X 0,Y 580.968,Z 534.976,A -85,B 0,C 180,E1 -1695.939,E2 -1695.939} C_VEL
LIN {X 0,Y 580.827,Z 548.921,A -85,B 0,C 180,E1 -1696.53,E2 -1696.53} C_VEL
LIN {X 0,Y 580.703,Z 560.448,A -85,B 0,C 180,E1 -1697.15,E2 -1697.15} C_VEL
LIN {X 0,Y 580.594,Z 571.263,A -85,B 0,C 180,E1 -1697.858,E2 -1697.858} C_VEL
LIN {X 0,Y 580.459,Z 582.359,A -85,B 0,C 180,E1 -1698.732,E2 -1698.732} C_VEL
LIN {X 0,Y 580.348,Z 592.668,A -85,B 0,C 180,E1 -1699.71,E2 -1699.71} C_VEL
LIN {X 0,Y 580.296,Z 601.835,A -85,B 0,C 180,E1 -1700.765,E2 -1700.765} C_VEL
LIN {X 0,Y 580.194,Z 609.473,A -85,B 0,C 180,E1 -1701.816,E2 -1701.816} C_VEL
LIN {X 0,Y 580.149,Z 614.882,A -85,B 0,C 180,E1 -1702.691,E2 -1702.691} C_VEL
LIN {X 0,Y 580.104,Z 620.31,A -85,B 0,C 180,E1 -1703.739,E2 -1703.739} C_VEL
LIN {X 0,Y 580.077,Z 624.769,A -85,B 0,C 180,E1 -1704.786,E2 -1704.786} C_VEL
LIN {X 0,Y 580.104,Z 628.312,A -85,B 0,C 180,E1 -1705.831,E2 -1705.831} C_VEL
LIN {X 0,Y 580.041,Z 631.722,A -85,B 0,C 180,E1 -1707.221,E2 -1707.221} C_VEL
LIN {X 0,Y 580.045,Z 633.764,A -85,B 0,C 180,E1 -1708.611,E2 -1708.611} C_VEL
LIN {X 0,Y 580.037,Z 634.496,A -85,B 0,C 180,E1 -1709.999,E2 -1709.999} C_VEL
LIN {X 0,Y 580.042,Z 633.867,A -85,B 0,C 180,E1 -1711.388,E2 -1711.388} C_VEL
LIN {X 0,Y 580.039,Z 631.901,A -85,B 0,C 180,E1 -1712.777,E2 -1712.777} C_VEL
LIN {X 0,Y 580.108,Z 630.437,A -85,B 0,C 180,E1 -1713.472,E2 -1713.472} C_VEL
LIN {X 0,Y 580.046,Z 626.347,A -85,B 0,C 180,E1 -1714.864,E2 -1714.864} C_VEL
LIN {X 0,Y 580.133,Z 622.309,A -85,B 0,C 180,E1 -1715.909,E2 -1715.909} C_VEL
LIN {X 0,Y 580.141,Z 617.294,A -85,B 0,C 180,E1 -1716.957,E2 -1716.957} C_VEL
LIN {X 0,Y 580.192,Z 610.065,A -85,B 0,C 180,E1 -1718.182,E2 -1718.182} C_VEL
LIN {X 0,Y 580.284,Z 602.545,A -85,B 0,C 180,E1 -1719.233,E2 -1719.233} C_VEL
LIN {X 0,Y 580.346,Z 593.515,A -85,B 0,C 180,E1 -1720.289,E2 -1720.289} C_VEL
LIN {X 0,Y 580.492,Z 582.511,A -85,B 0,C 180,E1 -1721.345,E2 -1721.345} C_VEL
LIN {X 0,Y 580.576,Z 571.306,A -85,B 0,C 180,E1 -1722.229,E2 -1722.229} C_VEL
LIN {X 0,Y 580.706,Z 560.495,A -85,B 0,C 180,E1 -1722.937,E2 -1722.937} C_VEL
LIN {X 0,Y 580.832,Z 548.973,A -85,B 0,C 180,E1 -1723.557,E2 -1723.557} C_VEL
LIN {X 0,Y 580.988,Z 535.891,A -85,B 0,C 180,E1 -1724.118,E2 -1724.118} C_VEL
LIN {X 0,Y 581.05,Z 521.737,A -85,B 0,C 180,E1 -1724.562,E2 -1724.562} C_VEL
LIN {X 0,Y 581.134,Z 508.442,A -85,B 0,C 180,E1 -1724.846,E2 -1724.846} C_VEL
LIN {X 0,Y 581.332,Z 376.54,A -85,B 0,C 180,E1 -1726.516,E2 -1726.516} C_VEL
LIN {X 0,Y 580.594,Z 372.223,A -85,B 0,C 180,E1 -1726.616,E2 -1726.616} C_VEL
LIN {X 0,Y 580.736,Z 352.888,A -85,B 0,C 180,E1 -1729.274,E2 -1729.274} C_VEL
LIN {X 0,Y 580.958,Z 332.104,A -85,B 0,C 180,E1 -1732.211,E2 -1732.211} C_VEL
LIN {X 0,Y 580.565,Z 328.18,A -85,B 0,C 180,E1 -1732.79,E2 -1732.79} C_VEL
LIN {X 0,Y 580.31,Z 326.958,A -85,B 0,C 180,E1 -1733.012,E2 -1733.012} C_VEL
LIN {X 0,Y 580.293,Z 326.824,A -85,B 0,C 180,E1 -1735.848,E2 -1735.848} C_VEL
LIN {X 0,Y 580.301,Z 326.827,A -85,B 0,C 180,E1 -1738.184,E2 -1738.184} C_VEL
LIN {X 0,Y 580.298,Z 326.823,A -85,B 0,C 180,E1 -1740.696,E2 -1740.696} C_VEL
LIN {X 0,Y 580.302,Z 326.819,A -85,B 0,C 180,E1 -1743.316,E2 -1743.316} C_VEL
LIN {X 0,Y 580.324,Z 326.822,A -85,B 0,C 180,E1 -1745.767,E2 -1745.767} C_VEL
LIN {X 0,Y 580.286,Z 326.829,A -85,B 0,C 180,E1 -1748.145,E2 -1748.145} C_VEL
LIN {X 0,Y 580.3,Z 326.819,A -85,B 0,C 180,E1 -1750.842,E2 -1750.842} C_VEL
LIN {X 0,Y 580.282,Z 326.828,A -85,B 0,C 180,E1 -1753.656,E2 -1753.656} C_VEL
LIN {X 0,Y 580.286,Z 326.821,A -85,B 0,C 180,E1 -1756.607,E2 -1756.607} C_VEL
LIN {X 0,Y 580.313,Z 326.819,A -85,B 0,C 180,E1 -1759.158,E2 -1759.158} C_VEL
LIN {X 0,Y 580.284,Z 326.825,A -85,B 0,C 180,E1 -1761.926,E2 -1761.926} C_VEL
LIN {X 0,Y 580.298,Z 326.82,A -85,B 0,C 180,E1 -1764.456,E2 -1764.456} C_VEL
LIN {X 0,Y 580.286,Z 326.823,A -85,B 0,C 180,E1 -1766.975,E2 -1766.975} C_VEL
LIN {X 0,Y 580.302,Z 326.825,A -85,B 0,C 180,E1 -1769.425,E2 -1769.425} C_VEL
LIN {X 0,Y 580.312,Z 326.817,A -85,B 0,C 180,E1 -1772.136,E2 -1772.136} C_VEL
LIN {X 0,Y 580.3,Z 326.821,A -85,B 0,C 180,E1 -1774.92,E2 -1774.92} C_VEL
LIN {X 0,Y 580.32,Z 326.823,A -85,B 0,C 180,E1 -1777.199,E2 -1777.199} C_VEL
LIN {X 0,Y 580.301,Z 326.82,A -85,B 0,C 180,E1 -1780.177,E2 -1780.177} C_VEL
LIN {X 0,Y 580.32,Z 326.823,A -85,B 0,C 180,E1 -1783.103,E2 -1783.103} C_VEL
LIN {X 0,Y 580.317,Z 326.818,A -85,B 0,C 180,E1 -1785.983,E2 -1785.983} C_VEL
LIN {X 0,Y 580.341,Z 326.818,A -85,B 0,C 180,E1 -1788.828,E2 -1788.828} C_VEL
LIN {X 0,Y 580.328,Z 326.819,A -85,B 0,C 180,E1 -1791.644,E2 -1791.644} C_VEL
LIN {X 0,Y 580.321,Z 326.818,A -85,B 0,C 180,E1 -1794.44,E2 -1794.44} C_VEL
LIN {X 0,Y 580.343,Z 326.821,A -85,B 0,C 180,E1 -1797.223,E2 -1797.223} C_VEL
LIN {X 0,Y 580.342,Z 326.814,A -85,B 0,C 180,E1 -1800,E2 -1800} C_VEL
LIN {X 0,Y 580.343,Z 326.82,A -85,B 0,C 180,E1 -1802.776,E2 -1802.776} C_VEL
LIN {X 0,Y 580.322,Z 326.818,A -85,B 0,C 180,E1 -1805.56,E2 -1805.56} C_VEL
LIN {X 0,Y 580.328,Z 326.818,A -85,B 0,C 180,E1 -1808.356,E2 -1808.356} C_VEL
LIN {X 0,Y 580.322,Z 326.82,A -85,B 0,C 180,E1 -1811.208,E2 -1811.208} C_VEL
LIN {X 0,Y 580.317,Z 326.818,A -85,B 0,C 180,E1 -1814.017,E2 -1814.017} C_VEL
LIN {X 0,Y 580.308,Z 326.825,A -85,B 0,C 180,E1 -1816.917,E2 -1816.917} C_VEL
LIN {X 0,Y 580.301,Z 326.819,A -85,B 0,C 180,E1 -1819.822,E2 -1819.822} C_VEL
LIN {X 0,Y 580.32,Z 326.824,A -85,B 0,C 180,E1 -1822.801,E2 -1822.801} C_VEL
LIN {X 0,Y 580.299,Z 326.821,A -85,B 0,C 180,E1 -1825.08,E2 -1825.08} C_VEL
LIN {X 0,Y 580.312,Z 326.817,A -85,B 0,C 180,E1 -1827.864,E2 -1827.864} C_VEL
LIN {X 0,Y 580.284,Z 326.826,A -85,B 0,C 180,E1 -1830.697,E2 -1830.697} C_VEL
LIN {X 0,Y 580.298,Z 326.82,A -85,B 0,C 180,E1 -1833.318,E2 -1833.318} C_VEL
LIN {X 0,Y 580.317,Z 326.819,A -85,B 0,C 180,E1 -1835.768,E2 -1835.768} C_VEL
LIN {X 0,Y 580.282,Z 326.826,A -85,B 0,C 180,E1 -1838.147,E2 -1838.147} C_VEL
LIN {X 0,Y 580.312,Z 326.82,A -85,B 0,C 180,E1 -1840.842,E2 -1840.842} C_VEL
LIN {X 0,Y 580.284,Z 326.823,A -85,B 0,C 180,E1 -1843.657,E2 -1843.657} C_VEL
LIN {X 0,Y 580.278,Z 326.825,A -85,B 0,C 180,E1 -1846.609,E2 -1846.609} C_VEL
LIN {X 0,Y 580.3,Z 326.819,A -85,B 0,C 180,E1 -1849.158,E2 -1849.158} C_VEL
LIN {X 0,Y 580.287,Z 326.829,A -85,B 0,C 180,E1 -1851.928,E2 -1851.928} C_VEL
LIN {X 0,Y 580.305,Z 326.822,A -85,B 0,C 180,E1 -1854.458,E2 -1854.458} C_VEL
LIN {X 0,Y 580.288,Z 326.821,A -85,B 0,C 180,E1 -1856.976,E2 -1856.976} C_VEL
LIN {X 0,Y 580.308,Z 326.822,A -85,B 0,C 180,E1 -1859.427,E2 -1859.427} C_VEL
LIN {X 0,Y 580.318,Z 326.824,A -85,B 0,C 180,E1 -1862.138,E2 -1862.138} C_VEL
LIN {X 0,Y 580.306,Z 326.821,A -85,B 0,C 180,E1 -1864.921,E2 -1864.921} C_VEL
LIN {X 0,Y 580.31,Z 327.103,A -85,B 0,C 180,E1 -1867.073,E2 -1867.073} C_VEL
LIN {X 0,Y 580.977,Z 331.79,A -85,B 0,C 180,E1 -1867.79,E2 -1867.79} C_VEL
LIN {X 0,Y 580.737,Z 352.565,A -85,B 0,C 180,E1 -1870.725,E2 -1870.725} C_VEL
LIN {X 0,Y 580.585,Z 372.227,A -85,B 0,C 180,E1 -1873.429,E2 -1873.429} C_VEL
LIN {X 0,Y 581.373,Z 377.488,A -85,B 0,C 180,E1 -1873.542,E2 -1873.542} C_VEL
LIN {X 0,Y 581.136,Z 509.937,A -85,B 0,C 180,E1 -1875.222,E2 -1875.222} C_VEL
LIN {X 0,Y 581.055,Z 524.292,A -85,B 0,C 180,E1 -1875.552,E2 -1875.552} C_VEL
LIN {X 0,Y 580.914,Z 537.732,A -85,B 0,C 180,E1 -1875.999,E2 -1875.999} C_VEL
LIN {X 0,Y 580.792,Z 551.662,A -85,B 0,C 180,E1 -1876.62,E2 -1876.62} C_VEL
LIN {X 0,Y 580.657,Z 564.116,A -85,B 0,C 180,E1 -1877.329,E2 -1877.329} C_VEL
LIN {X 0,Y 580.524,Z 576.653,A -85,B 0,C 180,E1 -1878.213,E2 -1878.213} C_VEL
LIN {X 0,Y 580.44,Z 587.901,A -85,B 0,C 180,E1 -1879.189,E2 -1879.189} C_VEL
LIN {X 0,Y 580.275,Z 597.859,A -85,B 0,C 180,E1 -1880.239,E2 -1880.239} C_VEL
LIN {X 0,Y 580.24,Z 606.178,A -85,B 0,C 180,E1 -1881.293,E2 -1881.293} C_VEL
LIN {X 0,Y 580.165,Z 614.132,A -85,B 0,C 180,E1 -1882.518,E2 -1882.518} C_VEL
LIN {X 0,Y 580.102,Z 620.531,A -85,B 0,C 180,E1 -1883.741,E2 -1883.741} C_VEL
LIN {X 0,Y 580.078,Z 624.964,A -85,B 0,C 180,E1 -1884.787,E2 -1884.787} C_VEL
LIN {X 0,Y 580.102,Z 628.447,A -85,B 0,C 180,E1 -1885.832,E2 -1885.832} C_VEL
LIN {X 0,Y 580.041,Z 631.835,A -85,B 0,C 180,E1 -1887.223,E2 -1887.223} C_VEL
LIN {X 0,Y 580.041,Z 633.834,A -85,B 0,C 180,E1 -1888.612,E2 -1888.612} C_VEL
LIN {X 0,Y 580.036,Z 634.5,A -85,B 0,C 180,E1 -1890.001,E2 -1890.001} C_VEL
LIN {X 0,Y 580.041,Z 633.831,A -85,B 0,C 180,E1 -1891.389,E2 -1891.389} C_VEL
LIN {X 0,Y 580.041,Z 631.83,A -85,B 0,C 180,E1 -1892.779,E2 -1892.779} C_VEL
LIN {X 0,Y 580.102,Z 628.44,A -85,B 0,C 180,E1 -1894.169,E2 -1894.169} C_VEL
LIN {X 0,Y 580.128,Z 623.565,A -85,B 0,C 180,E1 -1895.562,E2 -1895.562} C_VEL
LIN {X 0,Y 580.142,Z 617.048,A -85,B 0,C 180,E1 -1896.959,E2 -1896.959} C_VEL
LIN {X 0,Y 580.192,Z 609.794,A -85,B 0,C 180,E1 -1898.184,E2 -1898.184} C_VEL
LIN {X 0,Y 580.284,Z 600.816,A -85,B 0,C 180,E1 -1899.411,E2 -1899.411} C_VEL
LIN {X 0,Y 580.356,Z 591.383,A -85,B 0,C 180,E1 -1900.466,E2 -1900.466} C_VEL
LIN {X 0,Y 580.479,Z 581.31,A -85,B 0,C 180,E1 -1901.405,E2 -1901.405} C_VEL
LIN {X 0,Y 580.598,Z 569.421,A -85,B 0,C 180,E1 -1902.319,E2 -1902.319} C_VEL
LIN {X 0,Y 580.732,Z 556.63,A -85,B 0,C 180,E1 -1903.116,E2 -1903.116} C_VEL
LIN {X 0,Y 580.897,Z 544.142,A -85,B 0,C 180,E1 -1903.736,E2 -1903.736} C_VEL
LIN {X 0,Y 581.02,Z 531.159,A -85,B 0,C 180,E1 -1904.237,E2 -1904.237} C_VEL
LIN {X 0,Y 581.086,Z 517.139,A -85,B 0,C 180,E1 -1904.632,E2 -1904.632} C_VEL
LIN {X 0,Y 581.164,Z 502.544,A -85,B 0,C 180,E1 -1904.891,E2 -1904.891} C_VEL
LIN {X 0,Y 581.308,Z 376.451,A -85,B 0,C 180,E1 -1906.473,E2 -1906.473} C_VEL
LIN {X 0,Y 580.585,Z 372.2,A -85,B 0,C 180,E1 -1906.573,E2 -1906.573} C_VEL
LIN {X 0,Y 580.74,Z 352.557,A -85,B 0,C 180,E1 -1909.276,E2 -1909.276} C_VEL
LIN {X 0,Y 580.954,Z 331.776,A -85,B 0,C 180,E1 -1912.213,E2 -1912.213} C_VEL
LIN {X 0,Y 580.47,Z 327.853,A -85,B 0,C 180,E1 -1912.796,E2 -1912.796} C_VEL
LIN {X 0,Y 580.294,Z 326.905,A -85,B 0,C 180,E1 -1913.009,E2 -1913.009} C_VEL
LIN {X 0,Y 580.311,Z 326.82,A -85,B 0,C 180,E1 -1915.08,E2 -1915.08} C_VEL
LIN {X 0,Y 580.306,Z 326.825,A -85,B 0,C 180,E1 -1918.186,E2 -1918.186} C_VEL
LIN {X 0,Y 580.289,Z 326.824,A -85,B 0,C 180,E1 -1920.695,E2 -1920.695} C_VEL
LIN {X 0,Y 580.307,Z 326.82,A -85,B 0,C 180,E1 -1923.317,E2 -1923.317} C_VEL
LIN {X 0,Y 580.33,Z 326.822,A -85,B 0,C 180,E1 -1925.768,E2 -1925.768} C_VEL
LIN {X 0,Y 580.293,Z 326.829,A -85,B 0,C 180,E1 -1928.147,E2 -1928.147} C_VEL
LIN {X 0,Y 580.302,Z 326.82,A -85,B 0,C 180,E1 -1930.844,E2 -1930.844} C_VEL
LIN {X 0,Y 580.277,Z 326.829,A -85,B 0,C 180,E1 -1933.659,E2 -1933.659} C_VEL
LIN {X 0,Y 580.282,Z 326.823,A -85,B 0,C 180,E1 -1936.61,E2 -1936.61} C_VEL
LIN {X 0,Y 580.301,Z 326.822,A -85,B 0,C 180,E1 -1939.157,E2 -1939.157} C_VEL
LIN {X 0,Y 580.294,Z 326.828,A -85,B 0,C 180,E1 -1941.927,E2 -1941.927} C_VEL
LIN {X 0,Y 580.254,Z 326.827,A -85,B 0,C 180,E1 -1944.453,E2 -1944.453} C_VEL
LIN {X 0,Y 580.295,Z 326.822,A -85,B 0,C 180,E1 -1946.975,E2 -1946.975} C_VEL
LIN {X 0,Y 580.299,Z 326.828,A -85,B 0,C 180,E1 -1949.425,E2 -1949.425} C_VEL
LIN {X 0,Y 580.302,Z 326.823,A -85,B 0,C 180,E1 -1952.141,E2 -1952.141} C_VEL
LIN {X 0,Y 580.328,Z 327.007,A -85,B 0,C 180,E1 -1954.706,E2 -1954.706} C_VEL
LIN {X 0,Y 581.281,Z 332.573,A -85,B 0,C 180,E1 -1955.421,E2 -1955.421} C_VEL
LIN {X 0,Y 581.085,Z 352.828,A -85,B 0,C 180,E1 -1957.98,E2 -1957.98} C_VEL
LIN {X 0,Y 580.846,Z 374.642,A -85,B 0,C 180,E1 -1960.695,E2 -1960.695} C_VEL
LIN {X 0,Y 580.638,Z 397.317,A -85,B 0,C 180,E1 -1963.475,E2 -1963.475} C_VEL
LIN {X 0,Y 580.473,Z 420.903,A -85,B 0,C 180,E1 -1966.322,E2 -1966.322} C_VEL
LIN {X 0,Y 580.649,Z 422.619,A -85,B 0,C 180,E1 -1966.393,E2 -1966.393} C_VEL
LIN {X 0,Y 580.976,Z 431.551,A -85,B 0,C 180,E1 -1966.512,E2 -1966.512} C_VEL
LIN {X 0,Y 580.786,Z 530.366,A -85,B 0,C 180,E1 -1967.752,E2 -1967.752} C_VEL
LIN {X 0,Y 580.752,Z 543.733,A -85,B 0,C 180,E1 -1968.062,E2 -1968.062} C_VEL
LIN {X 0,Y 580.662,Z 556.958,A -85,B 0,C 180,E1 -1968.525,E2 -1968.525} C_VEL
LIN {X 0,Y 580.564,Z 568.931,A -85,B 0,C 180,E1 -1969.097,E2 -1969.097} C_VEL
LIN {X 0,Y 580.452,Z 580.339,A -85,B 0,C 180,E1 -1969.801,E2 -1969.801} C_VEL
LIN {X 0,Y 580.368,Z 590.605,A -85,B 0,C 180,E1 -1970.591,E2 -1970.591} C_VEL
LIN {X 0,Y 580.301,Z 599.882,A -85,B 0,C 180,E1 -1971.468,E2 -1971.468} C_VEL
LIN {X 0,Y 580.2,Z 608.851,A -85,B 0,C 180,E1 -1972.518,E2 -1972.518} C_VEL
LIN {X 0,Y 580.135,Z 616.505,A -85,B 0,C 180,E1 -1973.638,E2 -1973.638} C_VEL
LIN {X 0,Y 580.086,Z 622.664,A -85,B 0,C 180,E1 -1974.787,E2 -1974.787} C_VEL
LIN {X 0,Y 580.105,Z 627.021,A -85,B 0,C 180,E1 -1975.832,E2 -1975.832} C_VEL
LIN {X 0,Y 580.124,Z 629.322,A -85,B 0,C 180,E1 -1976.527,E2 -1976.527} C_VEL
LIN {X 0,Y 580.043,Z 631.193,A -85,B 0,C 180,E1 -1977.222,E2 -1977.222} C_VEL
LIN {X 0,Y 580.038,Z 632.628,A -85,B 0,C 180,E1 -1977.917,E2 -1977.917} C_VEL
LIN {X 0,Y 580.041,Z 634.254,A -85,B 0,C 180,E1 -1979.306,E2 -1979.306} C_VEL
LIN {X 0,Y 580.038,Z 634.496,A -85,B 0,C 180,E1 -1980,E2 -1980} C_VEL
LIN {X 0,Y 580.04,Z 634.314,A -85,B 0,C 180,E1 -1980.694,E2 -1980.694} C_VEL
LIN {X 0,Y 580.037,Z 632.771,A -85,B 0,C 180,E1 -1982.083,E2 -1982.083} C_VEL
LIN {X 0,Y 580.044,Z 631.412,A -85,B 0,C 180,E1 -1982.778,E2 -1982.778} C_VEL
LIN {X 0,Y 580.11,Z 628.539,A -85,B 0,C 180,E1 -1983.821,E2 -1983.821} C_VEL
LIN {X 0,Y 580.054,Z 624.64,A -85,B 0,C 180,E1 -1984.865,E2 -1984.865} C_VEL
LIN {X 0,Y 580.161,Z 619.608,A -85,B 0,C 180,E1 -1985.91,E2 -1985.91} C_VEL
LIN {X 0,Y 580.158,Z 613.271,A -85,B 0,C 180,E1 -1986.958,E2 -1986.958} C_VEL
LIN {X 0,Y 580.241,Z 605.37,A -85,B 0,C 180,E1 -1988.007,E2 -1988.007} C_VEL
LIN {X 0,Y 580.305,Z 597.299,A -85,B 0,C 180,E1 -1988.883,E2 -1988.883} C_VEL
LIN {X 0,Y 580.365,Z 587.46,A -85,B 0,C 180,E1 -1989.761,E2 -1989.761} C_VEL
LIN {X 0,Y 580.504,Z 576.402,A -85,B 0,C 180,E1 -1990.551,E2 -1990.551} C_VEL
LIN {X 0,Y 580.59,Z 565.585,A -85,B 0,C 180,E1 -1991.168,E2 -1991.168} C_VEL
LIN {X 0,Y 580.686,Z 552.841,A -85,B 0,C 180,E1 -1991.727,E2 -1991.727} C_VEL
LIN {X 0,Y 580.784,Z 539.752,A -85,B 0,C 180,E1 -1992.137,E2 -1992.137} C_VEL
LIN {X 0,Y 580.861,Z 526.218,A -85,B 0,C 180,E1 -1992.402,E2 -1992.402} C_VEL
LIN {X 0,Y 580.904,Z 480.85,A -85,B 0,C 180,E1 -1992.966,E2 -1992.966} C_VEL
LIN {X 0,Y 580.258,Z 475.045,A -85,B 0,C 180,E1 -1993.053,E2 -1993.053} C_VEL
LIN {X 0,Y 574.734,Z 456.353,A -85,B 0,C 180,E1 -1993.416,E2 -1993.416} C_VEL
